FUNCTION_BLOCK SM_TableManager EXTENDS  KvalStateMachineBaseExt IMPLEMENTS I_DoorTracker
VAR_INPUT
	pStatus_bAnyTableDoorTrackTargetChanged : POINTER TO BOOL;
	cmd_bReset							: BOOL; // reset from error state
	cmd_bAbort							: BOOL; // trigger event to abort any motion.
	// Job Sync (v1.0)
    fbJobSync							: FB_JobSynchronizer;
	cmd_sJobName 						: STRING;
	cmd_sJobNameLatched					: STRING;
	// commands
	cmd_bToFenceFwd						: BOOL;
	cmd_bToFenceRev						: BOOL;
	cmd_bCrossTransferFwd				: BOOL;
	cmd_bCrossTransferRev				: BOOL;
	cmd_bInlineTransferFwd				: BOOL;
	cmd_bInlineTransferRev				: BOOL;
	cmd_bJogSlow						: BOOL;
	cmd_bManualControlEnabled			: BOOL;
	cmd_bOutputPortEnabled				: BOOL;
	cmd_bRotate							: BOOL;
	cmd_bSelfCenter						: BOOL;	
	cmd_bExternal						: BOOL;
	cmd_bInternal						: BOOL;
	
	cmd_bDoorHasNoTarget 					: BOOL;
	cmd_bInitialized 						: BOOL;
	cmd_bDoorTransferInStarted 				: BOOL;
	cmd_bDoorDataReady 						: BOOL;
	cmd_bDoorDataReadyLatched 				: BOOL;
	cmd_bNewRouteRequested 					: BOOL;	
	cmd_bReroute							: BOOL;
	cmd_bReroutePending						: BOOL;
	cmd_bNewRouteRequestedFromDoorInMachineIdle : BOOL;
	cmd_bNewRouteRequestedFromWaitForFeedout : BOOL;
	cmd_bNewRouteRequestedFromAllTargetFeedoutPortsDisabled : BOOL;
	cmd_bNewRouteRequestedFromDoorHasNoTarget : BOOL;
	cmd_bNewRouteRequestedFromWaitingForClearRoute : BOOL;
	cmd_bDoorTransferInCompleted 			: BOOL;
	cmd_bFeedinStarted 						: BOOL;
	cmd_bFeedinCompleted 					: BOOL;

	cmd_bReadyToFeedOut : BOOL;
	cmd_bDoorTransferOutStartedFromIdle 	: BOOL;
	cmd_bDoorTransferOutStarted 			: BOOL;
	cmd_bDoorTransferOutCompleted 			: BOOL;
	cmd_bFeedoutStarted 					: BOOL;
	cmd_bFeedoutCompleted 					: BOOL;
	
	cmd_iSelectedDestinationIndexLast		: UINT;
	cmd_iSelectedDestinationIndex			: UINT;
	cmd_eIncomingDoorHand					: E_DOORHAND;
	cmd_eIncomingDoorHandLast				: E_DOORHAND;
	cmd_bIncomingDoorHandValid				: BOOL;
	cmd_iSelectedDestinationIndexLatched	: UINT;
	cmd_eIncomingDoorHandLatched			: E_DOORHAND;
	
	cmd_bNewTargetFeedoutPortSelected		: BOOL;
	cmd_stNewTargetFeedoutPort				: ST_FeedoutPort;
	config_bAutoDataReady					: BOOL; // true if table is an input port and the input port is configured for 'hungry-mode' where destination index 0 is mapped to 2 or more feed-out ports. 
													// On rising edge of LH/RH input valid, 'Data Ready' input is latched automatically, instead of user needs to press the 'Data Ready' button.
													// The physical 'Data Ready' button and the 'Destination Index' switch on the control box are not needed.
													
	config_bIsInputPortEnabled				: BOOL; // true if the table's input port is enabled and can receive door data from KvalCAM's job such as destination index and doorHand.
	config_bIsConveyorTable					: BOOL; // true if it's a conveyor table (class code 235); false = auto-cross transfer table (class code 234)
	config_bCanSelfCenter					: BOOL; // true if table has the self-centering option (Option S)
	config_bCanRotate						: BOOL; // true if table has the Auto-rotate option (Option A)
	cmd_bRequestNewRoute					: BOOL;
	config_bCanFeedinFromSideA				: BOOL; // true if it's an input port and its side A is available to feed-in door.
	config_bIsBufferTable					: BOOL; // true table is a T1 option, which can only do inline-transfer and not (cross-transfer or self-center)
	
	// --- Pointers to hot connect hardware --
	config_pstHcTransferTableHardware		: POINTER TO ST_HcTable;
	config_pstHcConveyorHardware			: POINTER TO ST_HcConveyor;
	
	// each table can have either a conveyor or a cross-and-straight manager, but not both.
	smC235FeedManager						: SM_235FeedManager; // manage cross feeding of the door in and out the machine.
	smC234FeedManager						: SM_234FeedManager; // manage cross-feeding of the door in and out the machine. 
	
	smDoorDasher							: SM_DoorDasher; // a door-dasher for DTS.
	
{IF defined (noHW) OR defined (noHW_UML)}
	psmHcFeedMotor							: POINTER TO SM_KMotorVFDEtherCATi550Ext; // balvm3539 1140 RPM 1/2 HP
{ELSE}
	psmHcFeedMotor							: POINTER TO SM_KMotorVFDEtherCATi550; // balvm3539 1140 RPM 1/2 HP
{END_IF}
	
	config_tRerouteWaitTime			: TIME := T#1.0S;
	
	// feed system configs
	// these are initialized from table topology sent by KvalCAM when press Ctrl+Shift+S key combination on the Main tab:
	config_iFeedFastSpeedFPM		: UINT := 150;				// Fast Feed Speed in Feet Per Minute
	config_iFeedSlowSpeedFPM		: UINT := 50;				// Slow Feed Speed in Feet Per Minute
	config_iFeedOutSpeedFPM			: UINT := 100;				// the speed at which the system feed's out.
	config_iCrossFeedFastSpeedFPM	: UINT := 75;				// Fast CrossFeed Speed in Feet Per Minute
	config_iCrossFeedSlowSpeedFPM	: UINT := 25;				// Slow CrossFeed Speed in Feet Per Minute
	config_iTableArrayIndex					: INT;						// The array table index.
	bDoorTrackDirty							: BOOL;
END_VAR
VAR_OUTPUT
	bTableReady : BOOL; // true if the table is ready to receive door.
	bTableIsEmpty : BOOL; // true if table is empty.
	bDoorInMachine				: BOOL; // true if NOT bTableIsEmpty AND door is completely inside machine (ie, not on C234's di_C or di_D eye)
	bOkToFeedOut		: BOOL;				// depending on the direction, is it ok to feed out?
	bHasDoor			: BOOL;		// true if bDoorInMachine is true.
	
	bReadyToRotate				: BOOL;
	bOkToSelfCenter : BOOL;
	bExternal: BOOL;
	status_bMoving		: BOOL;
	
	_bAllTargetFeedoutPortsDisabled : BOOL; // true if all of the Target's feedout ports are disabled.
	bAllTargetFeedoutPortsDisabled : BOOL; // true if all of the Target's feedout ports are disabled.
	_bDoorHasNoTarget : BOOL; // true if the init seq found a door on table but no Target is assigned.
	bDoorHasNoTarget : BOOL; // true if the init seq found a door on table but no Target is assigned.
	bCurrentTargetFeedoutPortEnabled : BOOL; // true if any of the Target's feed-out port is enabled.
	bAnyCurrentTargetFeedoutPortEnabled : BOOL;
	bAllCurrentTargetFeedoutPortsEnabled : BOOL;
	bAnySourceDestinationIndexFeedoutPortEnabled : BOOL;
	
	bAnyDestinationIndexFeedoutPortEnabled : BOOL; // true if any of the feed-out port is enabled from the DestinationIndexFeedoutPortsMapping.
	bDoorInMachineIdle : BOOL;
	bDoorWaitingForFeedOut: BOOL;
	bWaitForDataReadyOrTransferredIn : BOOL;
	bDoorTransferringIn : BOOL;
	bRouteReadyWaitForFeedIn : BOOL;
	bDoorFeedingIn : BOOL;
	bDoorFeedingOut : BOOL;
	bWaitAllTablesReady : BOOL;
	bWaitingForClearRoute: BOOL;
	bRequestNewRouteComplete : BOOL;
	bFindingPath: BOOL;
END_VAR
VAR CONSTANT
END_VAR
VAR_INPUT PERSISTENT
	stDoorTrack									: ST_DoorTrack;
END_VAR
VAR PERSISTENT
	config_bManualControlEnabled				: BOOL;
END_VAR
VAR
	tonEyeBlowoffTimer							: TON;
	tofJambKickOverTimer						: TOF;
	ftrigHasDoor								: F_TRIG;
	stDoorTrackLast								: ST_DoorTrack;
	rtrigPersistentDataChanged					: R_TRIG; // triggered when any of the persistent data (feedout aligned/manual control enabled/disabled changed)	
	rtrigAutofeedOn								: R_TRIG; // rising edge of cmd_bAutofeedOn.
	ftrigAutofeedOn								: F_TRIG; // falling edge of cmd_bAutofeedOn.		
	ftrigAnyChildNotAutofeedOn					: F_TRIG; // falling edge of cmd_bAutofeedOn.
	fbVfdSetupData								: FB_VfdSetupData;
	ftrigRotateComplete							: F_TRIG; // trigger to indicate the rotate sequence is completed.
	ftrigSelfCenterComplete						: F_TRIG; // trigger to indicate the self-center sequence is completed.
	rtrigExternal								: R_TRIG;
	rtrigInternal								: R_TRIG; 
	rtrigTargetFeedoutPortsDisabled				: R_TRIG; // On rising edge, all Target table's feed-out ports were turned off by operator. 
	ftrigTargetFeedoutPortsDisabled				: F_TRIG; // On falling edge, at least 1 of the table's feed-out ports was re-enabled or operator selected a new Target feed-out port. 
	rtrigAllTargetFeedoutPortsDisabled			: R_TRIG; // Door is in-machine. On rising edge, all Target's feedout ports are disabled.
	ftrigAllTargetFeedoutPortsDisabled			: F_TRIG; // Door is in-machine. On falling edge, at least one of Target's feedout ports is enabled.
	ftrigAnyNeighboringTableBusy				: F_TRIG;
	
	rtrigDoorHasNoTarget						: R_TRIG; // On rising edge, door is detected after init but has not Target set (ie, Target = -1). Might be data persistent is corrupted.
	ftrigDoorHasNoTarget						: F_TRIG; // On falling edge, door is assigned new Target by operator.
	
	ftrigSelectedDestinationIndexChanged		: F_TRIG;
	rtrigIncomingDoorHandChanged				: R_TRIG;
	ftrigIncomingDoorHandValid					: F_TRIG;
	rtrigAutoDataReadyChanged					: R_TRIG;
	
	rtrigRequestNewRoute						: R_TRIG; // on rising edge, set cmd_bNewRouteRequested:=true to filter out stDoorTrack.Target so it does not show up in the DestinationIndex popup.
	rtrigDoorDataReady							: R_TRIG; // On rising edge while waiting for feeding out or operator selected new feed-out port, a re-route is request.
	rtrigDoorDataReadyLatched					: R_TRIG;
	ftrigDoorDataReadyLatched					: F_TRIG;
	rtrigAnyFeedoutTableEmptyAndReady			: R_TRIG;
	rtrigAnyTableWithDoorInMachineAndIdle		: R_TRIG;
	
	ftrigDoorTransferredOut						: F_TRIG;
	rtrigTableIndexNotExistInDoorTrackTargetPath		: R_TRIG;
	
	rtrigAnyTableDoorTrackTargetChanged 		: R_TRIG;
	
	rtrigAllCurrentTargetFeedoutPortsEnabled	: R_TRIG;
	ftrigAllCurrentTargetFeedoutPortsEnabled	: F_TRIG;
	
	rtrigAnyCurrentTargetFeedoutPortEnabled 	: R_TRIG;
	ftrigAnyCurrentTargetFeedoutPortEnabled 	: F_TRIG;
	
	rtrigAnyDestinationIndexFeedoutPortEnabled 	: R_TRIG;
	ftrigAnyDestinationIndexFeedoutPortEnabled 	: F_TRIG;
	rtrigDoorDasherReady 						: R_TRIG; // rising edge the door is in-machine and is ready to be transferred out. 
	rtrigRerouteAllTablesWaitingTransferredOut  : R_TRIG;
	bReadyToFeedout								: BOOL;
	rtrigReadyToFeedout							: R_TRIG; 
	ftrigReadyToFeedout							: F_TRIG;
	ftrigAnyDoorDasherBusy						: F_TRIG;
	ftrigNewRouteRequestedFromAllTargetFeedoutPortsDisabled : F_TRIG;
	ftrigNewRouteRequestedFromDoorHasNoTarget 	: F_TRIG;
	
	iFeedFastSpeedRPM		: UINT;
	iFeedSlowSpeedRPM		: UINT;
	iFeedOutSpeedRPM		: UINT;
	iCrossFeedFastSpeedRPM	: UINT;
	iCrossFeedSlowSpeedRPM	: UINT;
	bHasTrackingInfo : BOOL;
	bHasEnabledFeedoutPorts : BOOL;
	bFoundValidRoute : BOOL;
	iSourceDestinationIndexFeedoutPortsCount : UINT;
	bIsHungryModeRouting : BOOL;	
	bAnyTableBusy : BOOL;
	bAllTablesReady : BOOL;	
	bAnyNeighboringTableHasDoorAndDataReadyActive : BOOL;
	bAnyFeedoutTableEmptyAndReady: BOOL;
	bAnyNeighboringTableEmpty: BOOL;
	bAnyTableEmpty : BOOL;
	bAnyTableWithDoorHasNoTarget : BOOL;
	bSelectedDestinationIndexChanged : BOOL;
    tofSelectedDestinationIndexChangedTimer : TOF;
	bAutoDataReadyConfigChanged : BOOL;
	bAutoDataReadyConfigLast : BOOL;
	
	tonAllTablesReady	: TON;
	rtrigAllTablesReady : R_TRIG;
END_VAR

{IF defined (noHW) OR defined (noHW_UML)}
	runMachine();
{ELSE}
	readInputs();
	runMachine();
	writeOutputs();
{END_IF}

METHOD addCandidateRouteToDoorTrack
VAR_INPUT
	pstCandidateRoute : POINTER TO ST_Route;
	eTargetFeedoutSide : E_FeedoutSideType;	
END_VAR
IF pstCandidateRoute = 0 THEN
	RETURN;
END_IF

// Commented out to include duplicate table indices. This is because each duplicate table index can have up to 3 different feed-out sides, each can have
// different OutfeedDoorOrientation. 
//IF NOT isTableIndexExistInCandidateRoutes(pstCandidateRoute^.TargetTableIndex) THEN
	stDoorTrack.CandidateRoutes.CandidateRoutes[stDoorTrack.CandidateRoutes.CandidateRoutesCount] := pstCandidateRoute^;
	stDoorTrack.CandidateRoutes.CandidateRoutes[stDoorTrack.CandidateRoutes.CandidateRoutesCount].TargetFeedoutSide := eTargetFeedoutSide;
	stDoorTrack.CandidateRoutes.CandidateRoutesCount := stDoorTrack.CandidateRoutes.CandidateRoutesCount + 1;
//END_IF
END_METHOD

METHOD addSearchResultToDoorTrack
VAR_INPUT
	searchResult : ST_SearchResult;
END_VAR
stDoorTrack.SearchResults.SearchResults[stDoorTrack.SearchResults.SearchResultsCount] := searchResult;
stDoorTrack.SearchResults.SearchResultsCount := stDoorTrack.SearchResults.SearchResultsCount + 1;
END_METHOD

METHOD addToAllEnabledFeedoutPorts
VAR_INPUT
	stFeedoutPort : ST_FeedoutPort;
END_VAR
IF stDoorTrack.AllEnabledFeedoutPorts.FeedoutPortsCount >= 0 AND
	stDoorTrack.AllEnabledFeedoutPorts.FeedoutPortsCount < MAX_FEEDOUT_PORTS THEN
	stDoorTrack.AllEnabledFeedoutPorts.FeedoutPorts[stDoorTrack.AllEnabledFeedoutPorts.FeedoutPortsCount] := stFeedoutPort;
	stDoorTrack.AllEnabledFeedoutPorts.FeedoutPortsCount := stDoorTrack.AllEnabledFeedoutPorts.FeedoutPortsCount + 1;
END_IF
END_METHOD

METHOD addToRejectedFeedoutPorts
VAR_INPUT
	stFeedoutPort : ST_FeedoutPort;
END_VAR
IF stDoorTrack.RejectedFeedoutPorts.FeedoutPortsCount >= 0 AND
	stDoorTrack.RejectedFeedoutPorts.FeedoutPortsCount < MAX_FEEDOUT_PORTS THEN
	stDoorTrack.RejectedFeedoutPorts.FeedoutPorts[stDoorTrack.RejectedFeedoutPorts.FeedoutPortsCount] := stFeedoutPort;
	stDoorTrack.RejectedFeedoutPorts.FeedoutPortsCount := stDoorTrack.RejectedFeedoutPorts.FeedoutPortsCount + 1;
END_IF
END_METHOD

METHOD addToReroutableFeedoutPorts
VAR_INPUT
	stFeedoutPort : ST_FeedoutPort;
END_VAR
IF stDoorTrack.ReroutableFeedoutPorts.FeedoutPortsCount >= 0 AND
	stDoorTrack.ReroutableFeedoutPorts.FeedoutPortsCount < MAX_SEARCH_RESULTS THEN
	stDoorTrack.ReroutableFeedoutPorts.FeedoutPorts[stDoorTrack.ReroutableFeedoutPorts.FeedoutPortsCount] := stFeedoutPort;
	stDoorTrack.ReroutableFeedoutPorts.FeedoutPortsCount := stDoorTrack.ReroutableFeedoutPorts.FeedoutPortsCount + 1;
END_IF
END_METHOD

METHOD addToTargetFeedoutPorts
VAR_INPUT
	stFeedoutPort : ST_FeedoutPort;
END_VAR
IF stDoorTrack.TargetFeedoutPorts.FeedoutPortsCount >= 0 AND
	stDoorTrack.TargetFeedoutPorts.FeedoutPortsCount < MAX_FEEDOUT_PORTS THEN
	stDoorTrack.TargetFeedoutPorts.FeedoutPorts[stDoorTrack.TargetFeedoutPorts.FeedoutPortsCount] := stFeedoutPort;
	stDoorTrack.TargetFeedoutPorts.FeedoutPortsCount := stDoorTrack.TargetFeedoutPorts.FeedoutPortsCount + 1;
END_IF
END_METHOD

METHOD allChildrenAutoFeedOn : BOOL
VAR_INPUT
END_VAR
IF config_bIsConveyorTable THEN
	allChildrenAutoFeedOn := smC235FeedManager.cmd_bAutoFeedOn AND smDoorDasher.cmd_bAutofeedOn;
ELSE
	allChildrenAutoFeedOn := smC234FeedManager.cmd_bAutoFeedOn AND smDoorDasher.cmd_bAutofeedOn;
END_IF
END_METHOD

METHOD allCurrentTargetFeedoutPortsEnabled : BOOL
VAR_INPUT
END_VAR
VAR
	i : INT;
	j : INT;
	k : INT;
	stFeedoutPort : ST_FeedoutPort;
END_VAR
allCurrentTargetFeedoutPortsEnabled := TRUE; // default true to only check after Target and DestinationIndex were assigned.
IF 	stDoorTrack.DestinationIndex <> -1 
	AND stDoorTrack.TargetFeedoutPorts.FeedoutPortsCount > 0 
	THEN		
	FOR i:=0 TO stDoorTrack.TargetFeedoutPorts.FeedoutPortsCount - 1 DO
		stFeedoutPort := stDoorTrack.TargetFeedoutPorts.FeedoutPorts[i];
		IF NOT MAIN.mainStateMachine.asmTableManagers[stFeedoutPort.TableIndex].isFeedoutSideEnabled(stFeedoutPort.Side) THEN
			allCurrentTargetFeedoutPortsEnabled := FALSE;
			RETURN;
		END_IF
	END_FOR
END_IF
END_METHOD

METHOD allTablesReady : BOOL
VAR 
	i : INT;
END_VAR
allTablesReady := TRUE;

FOR i:=0 TO  MAIN.mainStateMachine.smCtrlInterface.config_stTransferTableConfig.PrimaryTable.TablesCount-1 DO
	IF NOT MAIN.mainStateMachine.smCtrlInterface.config_stTransferTableConfig.PrimaryTable.Tables[i].IsFunctionalTable THEN
		CONTINUE;
	END_IF
	
	IF  MAIN.mainStateMachine.asmTableManagers[i].bDoorFeedingIn OR
		MAIN.mainStateMachine.asmTableManagers[i].bDoorFeedingOut OR
		MAIN.mainStateMachine.asmTableManagers[i].bDoorWaitingForFeedOut OR 
		(MAIN.mainStateMachine.asmTableManagers[i].bDoorInMachineIdle AND 
		MAIN.mainStateMachine.asmTableManagers[i].stDoorTrack.Target = i) THEN
		// door is at the Target feed-out port, skip checking.
		CONTINUE;
	END_IF
	
	IF MAIN.mainStateMachine.asmTableManagers[i].status_bBusy THEN
		allTablesReady := FALSE;
		RETURN;
	END_IF
END_FOR
END_METHOD

METHOD anyChildAutofeedOn : BOOL
VAR_INPUT
END_VAR
IF config_bIsConveyorTable THEN
	anyChildAutofeedOn :=   smC235FeedManager.cmd_bAutoFeedOn OR smDoorDasher.cmd_bAutofeedOn;
ELSE
	anyChildAutofeedOn :=   smC234FeedManager.cmd_bAutoFeedOn OR smDoorDasher.cmd_bAutofeedOn;
END_IF
END_METHOD

METHOD anyChildBusy : BOOL
VAR_INPUT
END_VAR
IF config_bIsConveyorTable THEN
	anyChildBusy := smC235FeedManager.status_bBusy;
ELSE
	anyChildBusy := smC234FeedManager.status_bBusy;
END_IF
END_METHOD

METHOD anyChildExternal : BOOL
VAR_INPUT
END_VAR
IF config_bIsConveyorTable THEN
	anyChildExternal :=   smC235FeedManager.bExternal;
ELSE
	anyChildExternal :=   smC234FeedManager.bExternal;
END_IF
END_METHOD

METHOD anyCurrentTargetFeedoutPortEnabled : BOOL
VAR_INPUT
END_VAR
VAR
	i : INT;
	j : INT;
	k : INT;
	stFeedoutPort : ST_FeedoutPort;
END_VAR
anyCurrentTargetFeedoutPortEnabled := FALSE;
IF 	stDoorTrack.DestinationIndex <> -1 
	AND stDoorTrack.TargetFeedoutPorts.FeedoutPortsCount > 0 
	THEN		
	FOR i:=0 TO stDoorTrack.TargetFeedoutPorts.FeedoutPortsCount - 1 DO
		stFeedoutPort := stDoorTrack.TargetFeedoutPorts.FeedoutPorts[i];
		IF MAIN.mainStateMachine.asmTableManagers[stFeedoutPort.TableIndex].isFeedoutSideEnabled(stFeedoutPort.Side) THEN
			anyCurrentTargetFeedoutPortEnabled := TRUE;
			RETURN;
		END_IF
	END_FOR
END_IF
END_METHOD

METHOD anyDestinationIndexFeedoutPortEnabled : BOOL
VAR_INPUT
END_VAR
VAR
	i : INT;
	j : INT;
	k : INT;
	stFeedoutPort : ST_FeedoutPort;
END_VAR
anyDestinationIndexFeedoutPortEnabled := TRUE; // default true to only check after Target and DestinationIndex were assigned.
IF 	stDoorTrack.DestinationIndex <> -1 
	THEN
	// the table has a Target table, now check if any of the feed-out port is enabled from the DestinationIndexFeedoutPortsMapping.
	anyDestinationIndexFeedoutPortEnabled := FALSE;
	i := stDoorTrack.Source;
	IF MAIN.mainStateMachine.smCtrlInterface.config_stTransferTableConfig.PrimaryTable.Tables[i].DestinationsFeedoutPortsMappingConfig.DestinationsFeedoutPortsMappingsCount > 0 THEN
		FOR j:=0 TO MAIN.mainStateMachine.smCtrlInterface.config_stTransferTableConfig.PrimaryTable.Tables[i].DestinationsFeedoutPortsMappingConfig.DestinationsFeedoutPortsMappingsCount - 1 DO
			IF MAIN.mainStateMachine.smCtrlInterface.config_stTransferTableConfig.PrimaryTable.Tables[i].DestinationsFeedoutPortsMappingConfig.DestinationsFeedoutPortsMappings[j].DestinationIndex = stDoorTrack.DestinationIndex THEN
				IF MAIN.mainStateMachine.smCtrlInterface.config_stTransferTableConfig.PrimaryTable.Tables[i].DestinationsFeedoutPortsMappingConfig.DestinationsFeedoutPortsMappings[j].FeedoutPortsCount > 0 THEN
					FOR k:=0 TO MAIN.mainStateMachine.smCtrlInterface.config_stTransferTableConfig.PrimaryTable.Tables[i].DestinationsFeedoutPortsMappingConfig.DestinationsFeedoutPortsMappings[j].FeedoutPortsCount - 1 DO
						stFeedoutPort := MAIN.mainStateMachine.smCtrlInterface.config_stTransferTableConfig.PrimaryTable.Tables[i].DestinationsFeedoutPortsMappingConfig.DestinationsFeedoutPortsMappings[j].FeedoutPorts[k];
						IF MAIN.mainStateMachine.asmTableManagers[stFeedoutPort.TableIndex].isFeedoutSideEnabled(stFeedoutPort.Side) THEN
							anyDestinationIndexFeedoutPortEnabled := TRUE;
							RETURN;
						END_IF
					END_FOR
				END_IF
				EXIT;
			END_IF
		END_FOR
	END_IF
END_IF
END_METHOD

METHOD anyDoorDasherBusy : bool
VAR 
	i : INT;
END_VAR
anyDoorDasherBusy := FALSE;	
FOR i:=0 TO MAIN.mainStateMachine.smCtrlInterface.config_stTransferTableConfig.PrimaryTable.TablesCount-1 DO
	IF NOT MAIN.mainStateMachine.smCtrlInterface.config_stTransferTableConfig.PrimaryTable.Tables[i].IsFunctionalTable THEN
		CONTINUE;
	END_IF
	IF MAIN.mainStateMachine.asmTableManagers[i].smDoorDasher.status_bBusy THEN
		anyDoorDasherBusy := TRUE;
		RETURN;		
	END_IF
END_FOR
END_METHOD

METHOD anyFeedoutTableEmptyAndReady : bool
VAR 
	i : INT;
END_VAR
anyFeedoutTableEmptyAndReady := FALSE;	
FOR i:=0 TO MAIN.mainStateMachine.smCtrlInterface.config_stTransferTableConfig.PrimaryTable.TablesCount-1 DO
	IF NOT (MAIN.mainStateMachine.smCtrlInterface.config_stTransferTableConfig.PrimaryTable.Tables[i].IsFunctionalTable AND
		MAIN.mainStateMachine.smCtrlInterface.config_stTransferTableConfig.PrimaryTable.Tables[i].IsOutputPort AND 
		MAIN.mainStateMachine.smCtrlInterface.config_stTransferTableConfig.PrimaryTable.Tables[i].OutputPortEnabled) THEN
		CONTINUE;
	END_IF
	IF  //MAIN.mainStateMachine.asmTableManagers[i].bWaitForDataReadyOrTransferredIn AND
		NOT (MAIN.mainStateMachine.asmTableManagers[i].bHasDoor OR 
			MAIN.mainStateMachine.asmTableManagers[i].status_bBusy OR
			MAIN.mainStateMachine.asmTableManagers[i].cmd_bDoorDataReadyLatched) THEN
		anyFeedoutTableEmptyAndReady := TRUE;
		RETURN;		
	END_IF
END_FOR
END_METHOD

METHOD anyNeighboringTableBusy : bool
VAR 
	northNeighborIndex : INT;
	southNeighborIndex : INT;
	eastNeighborIndex : INT;
	westNeighborIndex : INT;
END_VAR
anyNeighboringTableBusy := FALSE;
northNeighborIndex := MAIN.mainStateMachine.smCtrlInterface.config_stTransferTableConfig.PrimaryTable.Tables[config_iTableArrayIndex].NeighborNorthIndex;
southNeighborIndex := MAIN.mainStateMachine.smCtrlInterface.config_stTransferTableConfig.PrimaryTable.Tables[config_iTableArrayIndex].NeighborSouthIndex;
eastNeighborIndex := MAIN.mainStateMachine.smCtrlInterface.config_stTransferTableConfig.PrimaryTable.Tables[config_iTableArrayIndex].NeighborEastIndex;
westNeighborIndex := MAIN.mainStateMachine.smCtrlInterface.config_stTransferTableConfig.PrimaryTable.Tables[config_iTableArrayIndex].NeighborWestIndex;

IF northNeighborIndex <> -1 THEN
	IF MAIN.mainStateMachine.asmTableManagers[northNeighborIndex].status_bBusy THEN
		anyNeighboringTableBusy := TRUE;
		RETURN;
	END_IF
END_IF
IF southNeighborIndex <> -1 THEN
	IF MAIN.mainStateMachine.asmTableManagers[southNeighborIndex].status_bBusy THEN
		anyNeighboringTableBusy := TRUE;
		RETURN;
	END_IF
END_IF
IF eastNeighborIndex <> -1 THEN
	IF MAIN.mainStateMachine.asmTableManagers[eastNeighborIndex].status_bBusy THEN
		anyNeighboringTableBusy := TRUE;
		RETURN;
	END_IF
END_IF
IF westNeighborIndex <> -1 THEN
	IF MAIN.mainStateMachine.asmTableManagers[westNeighborIndex].status_bBusy THEN
		anyNeighboringTableBusy := TRUE;
		RETURN;
	END_IF
END_IF
END_METHOD

METHOD anyNeighboringTableEmpty : bool
VAR 
	northNeighborIndex : INT;
	southNeighborIndex : INT;
	eastNeighborIndex : INT;
	westNeighborIndex : INT;
END_VAR
anyNeighboringTableEmpty := FALSE;
northNeighborIndex := MAIN.mainStateMachine.smCtrlInterface.config_stTransferTableConfig.PrimaryTable.Tables[config_iTableArrayIndex].NeighborNorthIndex;
southNeighborIndex := MAIN.mainStateMachine.smCtrlInterface.config_stTransferTableConfig.PrimaryTable.Tables[config_iTableArrayIndex].NeighborSouthIndex;
eastNeighborIndex := MAIN.mainStateMachine.smCtrlInterface.config_stTransferTableConfig.PrimaryTable.Tables[config_iTableArrayIndex].NeighborEastIndex;
westNeighborIndex := MAIN.mainStateMachine.smCtrlInterface.config_stTransferTableConfig.PrimaryTable.Tables[config_iTableArrayIndex].NeighborWestIndex;

IF northNeighborIndex <> -1 THEN
	IF NOT (MAIN.mainStateMachine.asmTableManagers[northNeighborIndex].bHasDoor
			) THEN
		anyNeighboringTableEmpty := TRUE;
		RETURN;
	END_IF
END_IF
IF southNeighborIndex <> -1 THEN
	IF NOT (MAIN.mainStateMachine.asmTableManagers[southNeighborIndex].bHasDoor
			) THEN
		anyNeighboringTableEmpty := TRUE;
		RETURN;
	END_IF
END_IF
IF eastNeighborIndex <> -1 THEN
	IF NOT (MAIN.mainStateMachine.asmTableManagers[eastNeighborIndex].bHasDoor
			) THEN
		anyNeighboringTableEmpty := TRUE;
		RETURN;
	END_IF
END_IF
IF westNeighborIndex <> -1 THEN
	IF NOT (MAIN.mainStateMachine.asmTableManagers[westNeighborIndex].bHasDoor
			) THEN
		anyNeighboringTableEmpty := TRUE;
		RETURN;
	END_IF
END_IF
END_METHOD

METHOD anyNeighboringTableEmptyAndNotInPath : bool
VAR 
	northNeighborIndex : INT;
	southNeighborIndex : INT;
	eastNeighborIndex : INT;
	westNeighborIndex : INT;
END_VAR
anyNeighboringTableEmptyAndNotInPath := FALSE;
northNeighborIndex := MAIN.mainStateMachine.smCtrlInterface.config_stTransferTableConfig.PrimaryTable.Tables[config_iTableArrayIndex].NeighborNorthIndex;
southNeighborIndex := MAIN.mainStateMachine.smCtrlInterface.config_stTransferTableConfig.PrimaryTable.Tables[config_iTableArrayIndex].NeighborSouthIndex;
eastNeighborIndex := MAIN.mainStateMachine.smCtrlInterface.config_stTransferTableConfig.PrimaryTable.Tables[config_iTableArrayIndex].NeighborEastIndex;
westNeighborIndex := MAIN.mainStateMachine.smCtrlInterface.config_stTransferTableConfig.PrimaryTable.Tables[config_iTableArrayIndex].NeighborWestIndex;

IF northNeighborIndex <> -1 THEN
	IF NOT (MAIN.mainStateMachine.asmTableManagers[northNeighborIndex].bHasDoor
			 OR isNeighborInTargetPath(northNeighborIndex)
			) THEN
		anyNeighboringTableEmptyAndNotInPath := TRUE;
		RETURN;
	END_IF
END_IF
IF southNeighborIndex <> -1 THEN
	IF NOT (MAIN.mainStateMachine.asmTableManagers[southNeighborIndex].bHasDoor
			 OR isNeighborInTargetPath(southNeighborIndex)
			) THEN
		anyNeighboringTableEmptyAndNotInPath := TRUE;
		RETURN;
	END_IF
END_IF
IF eastNeighborIndex <> -1 THEN
	IF NOT (MAIN.mainStateMachine.asmTableManagers[eastNeighborIndex].bHasDoor
			 OR isNeighborInTargetPath(eastNeighborIndex)
			) THEN
		anyNeighboringTableEmptyAndNotInPath := TRUE;
		RETURN;
	END_IF
END_IF
IF westNeighborIndex <> -1 THEN
	IF NOT (MAIN.mainStateMachine.asmTableManagers[westNeighborIndex].bHasDoor
			 OR isNeighborInTargetPath(westNeighborIndex)
			) THEN
		anyNeighboringTableEmptyAndNotInPath := TRUE;
		RETURN;
	END_IF
END_IF
END_METHOD

METHOD anyNeighboringTableHasDoorAndDataReadyActive : bool
VAR 
	northNeighborIndex : INT;
	southNeighborIndex : INT;
	eastNeighborIndex : INT;
	westNeighborIndex : INT;
END_VAR
anyNeighboringTableHasDoorAndDataReadyActive := FALSE;
northNeighborIndex := MAIN.mainStateMachine.smCtrlInterface.config_stTransferTableConfig.PrimaryTable.Tables[config_iTableArrayIndex].NeighborNorthIndex;
southNeighborIndex := MAIN.mainStateMachine.smCtrlInterface.config_stTransferTableConfig.PrimaryTable.Tables[config_iTableArrayIndex].NeighborSouthIndex;
eastNeighborIndex := MAIN.mainStateMachine.smCtrlInterface.config_stTransferTableConfig.PrimaryTable.Tables[config_iTableArrayIndex].NeighborEastIndex;
westNeighborIndex := MAIN.mainStateMachine.smCtrlInterface.config_stTransferTableConfig.PrimaryTable.Tables[config_iTableArrayIndex].NeighborWestIndex;

IF northNeighborIndex <> -1 THEN
	IF (MAIN.mainStateMachine.asmTableManagers[northNeighborIndex].bHasDoor AND
		MAIN.mainStateMachine.asmTableManagers[northNeighborIndex].cmd_bDoorDataReadyLatched
			) THEN
		anyNeighboringTableHasDoorAndDataReadyActive := TRUE;
		RETURN;
	END_IF
END_IF
IF southNeighborIndex <> -1 THEN
	IF (MAIN.mainStateMachine.asmTableManagers[southNeighborIndex].bHasDoor AND
		MAIN.mainStateMachine.asmTableManagers[southNeighborIndex].cmd_bDoorDataReadyLatched
			) THEN
		anyNeighboringTableHasDoorAndDataReadyActive := TRUE;
		RETURN;
	END_IF
END_IF
IF eastNeighborIndex <> -1 THEN
	IF (MAIN.mainStateMachine.asmTableManagers[eastNeighborIndex].bHasDoor AND
		MAIN.mainStateMachine.asmTableManagers[eastNeighborIndex].cmd_bDoorDataReadyLatched
			) THEN
		anyNeighboringTableHasDoorAndDataReadyActive := TRUE;
		RETURN;
	END_IF
END_IF
IF westNeighborIndex <> -1 THEN
	IF (MAIN.mainStateMachine.asmTableManagers[westNeighborIndex].bHasDoor AND
		MAIN.mainStateMachine.asmTableManagers[westNeighborIndex].cmd_bDoorDataReadyLatched
			) THEN
		anyNeighboringTableHasDoorAndDataReadyActive := TRUE;
		RETURN;
	END_IF
END_IF
END_METHOD

METHOD anySourceDestinationIndexFeedoutPortEnabled : BOOL
VAR_INPUT
	selectedDestinationIndex : INT;
END_VAR
VAR
	j : INT;
	k : INT;
	stFeedoutPort : ST_FeedoutPort;
END_VAR
anySourceDestinationIndexFeedoutPortEnabled := FALSE; 
IF MAIN.mainStateMachine.smCtrlInterface.config_stTransferTableConfig.PrimaryTable.Tables[config_iTableArrayIndex].DestinationsFeedoutPortsMappingConfig.DestinationsFeedoutPortsMappingsCount > 0 THEN
	FOR j:=0 TO MAIN.mainStateMachine.smCtrlInterface.config_stTransferTableConfig.PrimaryTable.Tables[config_iTableArrayIndex].DestinationsFeedoutPortsMappingConfig.DestinationsFeedoutPortsMappingsCount - 1 DO
		IF MAIN.mainStateMachine.smCtrlInterface.config_stTransferTableConfig.PrimaryTable.Tables[config_iTableArrayIndex].DestinationsFeedoutPortsMappingConfig.DestinationsFeedoutPortsMappings[j].FeedoutPortsCount > 0 THEN
			FOR k:=0 TO MAIN.mainStateMachine.smCtrlInterface.config_stTransferTableConfig.PrimaryTable.Tables[config_iTableArrayIndex].DestinationsFeedoutPortsMappingConfig.DestinationsFeedoutPortsMappings[j].FeedoutPortsCount - 1 DO
				IF MAIN.mainStateMachine.smCtrlInterface.config_stTransferTableConfig.PrimaryTable.Tables[config_iTableArrayIndex].DestinationsFeedoutPortsMappingConfig.DestinationsFeedoutPortsMappings[j].DestinationIndex = selectedDestinationIndex THEN
					stFeedoutPort := MAIN.mainStateMachine.smCtrlInterface.config_stTransferTableConfig.PrimaryTable.Tables[config_iTableArrayIndex].DestinationsFeedoutPortsMappingConfig.DestinationsFeedoutPortsMappings[j].FeedoutPorts[k];
					IF MAIN.mainStateMachine.asmTableManagers[stFeedoutPort.TableIndex].isFeedoutSideEnabled(stFeedoutPort.Side) THEN
						anySourceDestinationIndexFeedoutPortEnabled := TRUE;
						RETURN;
					END_IF
				END_IF
			END_FOR
		END_IF
	END_FOR
END_IF
END_METHOD

METHOD anyTableBusy : BOOL
VAR 
	i : INT;
END_VAR
anyTableBusy := FALSE;

FOR i:=0 TO  MAIN.mainStateMachine.smCtrlInterface.config_stTransferTableConfig.PrimaryTable.TablesCount-1 DO
	IF NOT MAIN.mainStateMachine.smCtrlInterface.config_stTransferTableConfig.PrimaryTable.Tables[i].IsFunctionalTable THEN
		CONTINUE;
	END_IF
	
	IF MAIN.mainStateMachine.asmTableManagers[i].status_bBusy THEN
		anyTableBusy := TRUE;
		RETURN;
	END_IF
END_FOR
END_METHOD

METHOD anyTableEmpty : BOOL
VAR 
	i : INT;
END_VAR
anyTableEmpty := FALSE;

FOR i:=0 TO  MAIN.mainStateMachine.smCtrlInterface.config_stTransferTableConfig.PrimaryTable.TablesCount-1 DO
	IF NOT MAIN.mainStateMachine.smCtrlInterface.config_stTransferTableConfig.PrimaryTable.Tables[i].IsFunctionalTable THEN
		CONTINUE;
	END_IF
	
	IF NOT MAIN.mainStateMachine.asmTableManagers[i].bHasDoor THEN
		anyTableEmpty := TRUE;
		RETURN;
	END_IF
END_FOR
END_METHOD

METHOD anyTableWithDoorHasNoTarget : BOOL
VAR 
	i : INT;
END_VAR
anyTableWithDoorHasNoTarget := FALSE;

FOR i:=0 TO MAIN.mainStateMachine.smCtrlInterface.config_stTransferTableConfig.PrimaryTable.TablesCount-1 DO
	IF NOT (MAIN.mainStateMachine.smCtrlInterface.config_stTransferTableConfig.PrimaryTable.Tables[i].IsFunctionalTable) THEN
		CONTINUE;
	END_IF
	IF MAIN.mainStateMachine.asmTableManagers[i].bDoorHasNoTarget THEN
		anyTableWithDoorHasNoTarget := TRUE;
		RETURN;
	END_IF
END_FOR
END_METHOD

METHOD autofeedOff
VAR_INPUT
END_VAR
smC234FeedManager.cmd_bAutoFeedOn := FALSE;
smC235FeedManager.cmd_bAutoFeedOn := FALSE;
smC234FeedManager.cmd_bAbort := TRUE;
smC235FeedManager.cmd_bAbort := TRUE;
smDoorDasher.cmd_bAutofeedOn := FALSE;
END_METHOD

METHOD autofeedOn
VAR_INPUT
END_VAR
smC234FeedManager.cmd_bAutoFeedOn := TRUE;
smC235FeedManager.cmd_bAutoFeedOn := TRUE;
smDoorDasher.cmd_bAutofeedOn := TRUE;
END_METHOD

METHOD blinkReadyToFeedoutSideA
VAR_INPUT
END_VAR
IF config_bIsConveyorTable THEN
	;
ELSE
	smC234FeedManager.blinkReadyToFeedoutSideA();
END_IF
END_METHOD

METHOD blinkReadyToFeedoutSideB
VAR_INPUT
END_VAR
IF config_bIsConveyorTable THEN
	;
ELSE
	smC234FeedManager.blinkReadyToFeedoutSideB();
END_IF
END_METHOD

METHOD blinkReadyToFeedoutSideC
VAR_INPUT
END_VAR
IF config_bIsConveyorTable THEN
	smC235FeedManager.blinkReadyToFeedoutSideC();
ELSE
	smC234FeedManager.blinkReadyToFeedoutSideC();
END_IF
END_METHOD

METHOD blinkReadyToFeedoutSideD
VAR_INPUT
END_VAR
IF config_bIsConveyorTable THEN
	smC235FeedManager.blinkReadyToFeedoutSideD();
ELSE
	smC234FeedManager.blinkReadyToFeedoutSideD();
END_IF
END_METHOD

METHOD blinkReadyToFeedoutSides
VAR_INPUT	
END_VAR
VAR 
	i : INT;
END_VAR
FOR i:=0 TO stDoorTrack.TargetFeedoutPorts.FeedoutPortsCount -1 DO
	IF stDoorTrack.TargetFeedoutPorts.FeedoutPorts[i].Side = E_FeedoutSideType.A THEN
		blinkReadyToFeedoutSideA();
	ELSIF stDoorTrack.TargetFeedoutPorts.FeedoutPorts[i].Side = E_FeedoutSideType.B THEN
		blinkReadyToFeedoutSideB();
	ELSIF stDoorTrack.TargetFeedoutPorts.FeedoutPorts[i].Side = E_FeedoutSideType.C THEN
		blinkReadyToFeedoutSideC();
	ELSIF stDoorTrack.TargetFeedoutPorts.FeedoutPorts[i].Side = E_FeedoutSideType.D THEN
		blinkReadyToFeedoutSideD();
	END_IF
END_FOR
END_METHOD

METHOD clearDoorTrack
VAR_INPUT
END_VAR
IF config_bNoHardwareTestMode THEN
	smC234FeedManager.di_InMachineEye := FALSE;
END_IF
stDoorTrack := stDoorTrackDefault;
stDoorTrackLast := stDoorTrackDefault;
setTableEmptyStatus(TRUE);
END_METHOD

METHOD clearDoorTrackDoorIdAndTarget
VAR_INPUT
END_VAR
stDoorTrack.DoorId := 0;
stDoorTrack.Target := -1;
stDoorTrack.TargetName := '--';
stDoorTrack.DoorRotateRequired := FALSE;
stDoorTrack.DoorWasRotated := FALSE;
stDoorTrack.DoorIsRotating := FALSE;
END_METHOD

METHOD clearLastError
VAR 
	i : INT;
END_VAR
SUPER^.clearLastError();
smC234FeedManager.clearLastError();
smC235FeedManager.clearLastError();
smDoorDasher.clearLastError();
END_METHOD

METHOD clearNextDoorId
VAR_INPUT	
END_VAR
stDoorTrack.DoorId := 0;
END_METHOD

METHOD computeDirectionalChanges : INT
VAR_INPUT
	pstPath : POINTER TO ST_PathInfo;
END_VAR
VAR
	i : INT;
	directionalChanges : INT;
	curDirection : E_Direction;
	tempDirection : E_Direction;
END_VAR
IF pstPath = 0 THEN
	computeDirectionalChanges := MAX_INT;
	RETURN;
END_IF

IF pstPath^.PathCount <= 1 THEN
	computeDirectionalChanges := 0;
	RETURN;
END_IF

curDirection := pstPath^.Path[0].Direction;

FOR i:=1 TO pstPath^.PathCount - 1 DO
	tempDirection := pstPath^.Path[i].Direction;
	IF tempDirection <> E_Direction.None AND curDirection <> tempDirection THEN
		curDirection := tempDirection;
		directionalChanges := directionalChanges + 1;
	END_IF
	
END_FOR

computeDirectionalChanges := directionalChanges;
END_METHOD

METHOD computeDoorsInPath : INT
VAR_INPUT
	pstPath : POINTER TO ST_PathInfo;
END_VAR
VAR
	i : INT;
	doorsInPath : INT;
END_VAR
IF pstPath = 0 THEN
	computeDoorsInPath := MAX_INT;
	RETURN;
END_IF

FOR i:= 0 TO pstPath^.PathCount - 1 DO
	IF MAIN.mainStateMachine.asmTableManagers[pstPath^.Path[i].TableIndex].bHasDoor THEN
		doorsInPath := doorsInPath + 1;
	END_IF
END_FOR

computeDoorsInPath := doorsInPath;
END_METHOD

// compute the score for each of the search result. The result with highest final score is selected and its target is saved in DoorTrack.Target.
METHOD computeFinalScore
VAR
	numberOfHopsWeight : LREAL;
	directionChangesWeight : LREAL;
	doorsInPathWeight : LREAL;
	numberOfHopsMin : LREAL;
	directionChangesMin : LREAL;
	doorsInPathMin : LREAL;
	hasEmptyTableInPathWeight : LREAL;
	hasIncomingDoorInPathWeight : LREAL;
	pstSearchResults : POINTER TO ST_SearchResults;
	pstSearchResult : POINTER TO ST_SearchResult;
	pstPathInfo : pointer to ST_PathInfo;
	pstSearchResultWithMaxFinalScore : POINTER TO ST_SearchResult;
	i : INT;
	target : INT;
	stRejectedFeedoutPort : ST_FeedoutPort;
	stReroutableFeedoutPort : ST_FeedoutPort;
	stTargetFeedoutPorts : ST_FeedoutPortsConfig;
	stAllEnabledFeedoutPorts : ST_FeedoutPortsConfig;
	stRejectedFeedoutPorts : ST_FeedoutPortsConfig;
	stReroutableFeedoutPorts : ST_ReroutableFeedoutPortsConfig;
	stCandidateRoutes : ST_CandidateRoutes;
	stSearchResults : ST_SearchResults;
END_VAR
pstSearchResults := ADR(stDoorTrack.SearchResults);
numberOfHopsWeight := MAIN.mainStateMachine.smCtrlInterface.config_stTransferTableConfig.PrimaryTable.PathFindingConfig.NumberHopsWeight;
directionChangesWeight := MAIN.mainStateMachine.smCtrlInterface.config_stTransferTableConfig.PrimaryTable.PathFindingConfig.DirectionalChangesWeight;
doorsInPathWeight := MAIN.mainStateMachine.smCtrlInterface.config_stTransferTableConfig.PrimaryTable.PathFindingConfig.DoorsInPathWeight;
hasEmptyTableInPathWeight := MAIN.mainStateMachine.smCtrlInterface.config_stTransferTableConfig.PrimaryTable.PathFindingConfig.HasEmptyTableInPathWeight;
hasIncomingDoorInPathWeight := MAIN.mainStateMachine.smCtrlInterface.config_stTransferTableConfig.PrimaryTable.PathFindingConfig.HasIncomingDoorInPathWeight;
stDoorTrack.RejectedFeedoutPorts.FeedoutPortsCount := 0; // Reset to 0 for counting the rejected feed-out ports for re-routing.
stDoorTrack.ReroutableFeedoutPorts.FeedoutPortsCount := 0; // Reset to 0 for counting the reroutable feed-out ports for re-routing.
bFoundValidRoute := FALSE;

FOR i := 0 TO pstSearchResults^.SearchResultsCount -1 DO
	pstSearchResult := ADR(pstSearchResults^.SearchResults[i]);
	pstPathInfo := ADR(pstSearchResult^.PathIno);
	pstSearchResult^.NumberOfHops := pstSearchResult^.PathIno.PathCount;
	pstSearchResult^.DirectionalChanges := computeDirectionalChanges(pstPathInfo);
	pstSearchResult^.DoorsInPath := computeDoorsInPath(pstPathInfo);
	pstSearchResult^.HasEmptyTableInPath := hasEmptyTableInPath(pstPathInfo);
	pstSearchResult^.HasDoorGoingOppositeDirection := hasDoorGoingOppositeDirection(pstPathInfo);
	pstSearchResult^.HasIncomingDoorInPath := hasIncomingDoorInPath(pstPathInfo);
	pstSearchResult^.HasDeadlockedDoorInPath := hasDeadlockedDoorInPath(pstPathInfo);
	pstSearchResult^.RotationRequired := doesPathRequireRotation(pstPathInfo, stDoorTrack.Source, stDoorTrack.DoorHand, pstSearchResult^.TargetFeedoutSide);
	pstSearchResult^.PathHasRotateOption := pathHasRotateOption(pstPathInfo);
END_FOR

numberOfHopsMin := minNumberOfHops(pstSearchResults);
directionChangesMin := minDirectionalChanges(pstSearchResults);
doorsInPathMin := minDoorsInPath(pstSearchResults);

FOR i := 0 TO pstSearchResults^.SearchResultsCount -1 DO
	pstSearchResult := ADR(pstSearchResults^.SearchResults[i]);
	
	pstSearchResult^.NumberOfHopsSubScore := numberOfHopsMin / pstSearchResult^.NumberOfHops * numberOfHopsWeight;
	
	IF pstSearchResult^.DirectionalChanges = 0 THEN
		pstSearchResult^.DirectionChangesSubScore := directionChangesWeight;
	ELSE
		pstSearchResult^.DirectionChangesSubScore := directionChangesMin / pstSearchResult^.DirectionalChanges * directionChangesWeight;
	END_IF
	
	IF pstSearchResult^.DoorsInPath = 0 THEN
		pstSearchResult^.DoorsInPathSubScore :=  doorsInPathWeight;
	ELSE
		pstSearchResult^.DoorsInPathSubScore :=  doorsInPathMin / pstSearchResult^.DoorsInPath * doorsInPathWeight;
	END_IF
 
	pstSearchResult^.HasEmptyTableInPathSubScore :=  BOOL_TO_INT(pstSearchResult^.HasEmptyTableInPath) * hasEmptyTableInPathWeight;
	
	pstSearchResult^.HasIncomingDoorInPathSubScore :=  BOOL_TO_INT(pstSearchResult^.HasIncomingDoorInPath) * hasIncomingDoorInPathWeight;
	
	pstSearchResult^.FinalScore := pstSearchResult^.NumberOfHopsSubScore + pstSearchResult^.DirectionChangesSubScore + pstSearchResult^.DoorsInPathSubScore + pstSearchResult^.HasEmptyTableInPathSubScore + pstSearchResult^.HasIncomingDoorInPathSubScore;
	
	IF pstSearchResult^.HasDoorGoingOppositeDirection OR
		pstSearchResult^.HasDeadlockedDoorInPath OR		
		((pstSearchResult^.RotationRequired XOR stDoorTrackLast.DoorWasRotated) AND NOT pstSearchResult^.PathHasRotateOption) 
	THEN
		IF cmd_bRequestNewRoute THEN
			stRejectedFeedoutPort.TableIndex := pstSearchResult^.PathIno.Path[pstSearchResult^.PathIno.PathCount - 1].TableIndex;
			stRejectedFeedoutPort.Side := pstSearchResult^.TargetFeedoutSide;
			addToRejectedFeedoutPorts(stRejectedFeedoutPort);
		END_IF
		CONTINUE;
	END_IF
	
	IF cmd_bRequestNewRoute THEN
		stReroutableFeedoutPort.TableIndex := pstSearchResult^.PathIno.Path[pstSearchResult^.PathIno.PathCount - 1].TableIndex;
		stReroutableFeedoutPort.Side := pstSearchResult^.TargetFeedoutSide;
		addToReroutableFeedoutPorts(stReroutableFeedoutPort);
	ELSE 	
		IF pstSearchResultWithMaxFinalScore = 0 THEN
			pstSearchResultWithMaxFinalScore := pstSearchResult;
		ELSIF pstSearchResult^.FinalScore > pstSearchResultWithMaxFinalScore^.FinalScore THEN
			pstSearchResultWithMaxFinalScore := pstSearchResult;
		END_IF
	END_IF
END_FOR

IF cmd_bRequestNewRoute THEN
	// save these before restoring to last door-track.	
	stAllEnabledFeedoutPorts := stDoorTrack.AllEnabledFeedoutPorts;
	stRejectedFeedoutPorts := stDoorTrack.RejectedFeedoutPorts;
	stReroutableFeedoutPorts := stDoorTrack.ReroutableFeedoutPorts;
	stCandidateRoutes := stDoorTrack.CandidateRoutes;
	stSearchResults := stDoorTrack.SearchResults;
	
	// restore to last door track. 
	stDoorTrack := stDoorTrackLast;
	
	// restore these for oeprator's manual rerouting.
	stDoorTrack.AllEnabledFeedoutPorts := stAllEnabledFeedoutPorts;
	stDoorTrack.RejectedFeedoutPorts := stRejectedFeedoutPorts;
	stDoorTrack.ReroutableFeedoutPorts := stReroutableFeedoutPorts;	
	stDoorTrack.CandidateRoutes := stCandidateRoutes;
	stDoorTrack.SearchResults := stSearchResults;
ELSE	
	IF pstSearchResultWithMaxFinalScore <> 0 THEN
		IF pstSearchResultWithMaxFinalScore^.PathIno.PathCount > 0 THEN
			stDoorTrack.Target := pstSearchResultWithMaxFinalScore^.PathIno.Path[pstSearchResultWithMaxFinalScore^.PathIno.PathCount - 1].TableIndex;
			stDoorTrack.TargetName := MAIN.mainStateMachine.smCtrlInterface.config_stTransferTableConfig.PrimaryTable.Tables[stDoorTrack.Target].Name;
			stDoorTrack.TargetPath := pstSearchResultWithMaxFinalScore^.PathIno;
			stDoorTrack.TargetFeedoutSide := pstSearchResultWithMaxFinalScore^.TargetFeedoutSide;
			stDoorTrack.DoorRotateRequired := pstSearchResultWithMaxFinalScore^.RotationRequired;
			stDoorTrack.DoorWasRotated := stDoorTrackLast.DoorWasRotated;
			stDoorTrack.HasEmptyTableInPath := pstSearchResultWithMaxFinalScore^.HasEmptyTableInPath;
			stDoorTrack.HasDoorGoingOppositeDirection := pstSearchResultWithMaxFinalScore^.HasDoorGoingOppositeDirection;
			stDoorTrack.HasIncomingDoorInPath := pstSearchResultWithMaxFinalScore^.HasIncomingDoorInPath;
			stDoorTrack.HasDeadlockedDoorInPath := pstSearchResultWithMaxFinalScore^.HasDeadlockedDoorInPath;
		END_IF
	ELSE
		// Failed to find new route. Set to default to clear TargetDoorTrackInfo on HMI.
		stDoorTrack := stDoorTrackDefault;
	END_IF
END_IF

IF cmd_bNewRouteRequestedFromDoorHasNoTarget AND stDoorTrack.Target = -1 THEN
	stDoorTrack.TargetFeedoutPorts := stAllEnabledFeedoutPorts;
ELSE
	bFoundValidRoute := stDoorTrack.Target <> -1 AND stDoorTrack.TargetPath.PathCount > 0;
	IF NOT bFoundValidRoute THEN
		stTargetFeedoutPorts := stDoorTrack.TargetFeedoutPorts;
		// restore to last door track. 
		stDoorTrack := stDoorTrackLast;		
		stDoorTrack.TargetFeedoutPorts := stTargetFeedoutPorts;
	END_IF
END_IF
END_METHOD

METHOD currentTargetFeedoutPortEnabled : BOOL
VAR_INPUT
END_VAR
VAR
	i : INT;
	j : INT;
	k : INT;
	stFeedoutPort : ST_FeedoutPort;
END_VAR
currentTargetFeedoutPortEnabled := TRUE; // default true to only check after Target and DestinationIndex were assigned.
IF 	stDoorTrack.DestinationIndex <> -1 THEN
	// the table has a Target table, now check if any of the feed-out port is enabled.
	currentTargetFeedoutPortEnabled := FALSE;
	i := stDoorTrack.Source;
	IF MAIN.mainStateMachine.smCtrlInterface.config_stTransferTableConfig.PrimaryTable.Tables[i].DestinationsFeedoutPortsMappingConfig.DestinationsFeedoutPortsMappingsCount > 0 THEN
		FOR j:=0 TO MAIN.mainStateMachine.smCtrlInterface.config_stTransferTableConfig.PrimaryTable.Tables[i].DestinationsFeedoutPortsMappingConfig.DestinationsFeedoutPortsMappingsCount - 1 DO
			IF MAIN.mainStateMachine.smCtrlInterface.config_stTransferTableConfig.PrimaryTable.Tables[i].DestinationsFeedoutPortsMappingConfig.DestinationsFeedoutPortsMappings[j].DestinationIndex = stDoorTrack.DestinationIndex THEN
				IF MAIN.mainStateMachine.smCtrlInterface.config_stTransferTableConfig.PrimaryTable.Tables[i].DestinationsFeedoutPortsMappingConfig.DestinationsFeedoutPortsMappings[j].FeedoutPortsCount > 0 THEN
					FOR k:=0 TO MAIN.mainStateMachine.smCtrlInterface.config_stTransferTableConfig.PrimaryTable.Tables[i].DestinationsFeedoutPortsMappingConfig.DestinationsFeedoutPortsMappings[j].FeedoutPortsCount - 1 DO
						stFeedoutPort := MAIN.mainStateMachine.smCtrlInterface.config_stTransferTableConfig.PrimaryTable.Tables[i].DestinationsFeedoutPortsMappingConfig.DestinationsFeedoutPortsMappings[j].FeedoutPorts[k];
						IF stDoorTrack.Target = stFeedoutPort.TableIndex AND 
							stDoorTrack.TargetFeedoutSide = stFeedoutPort.Side AND 
							MAIN.mainStateMachine.asmTableManagers[stFeedoutPort.TableIndex].isFeedoutSideEnabled(stFeedoutPort.Side) THEN
							currentTargetFeedoutPortEnabled := TRUE;
							RETURN;
						END_IF
					END_FOR
				END_IF
				EXIT;
			END_IF
		END_FOR
	END_IF
END_IF
END_METHOD

METHOD doesPathRequireRotation : BOOL
VAR_INPUT
	pstPath : POINTER TO ST_PathInfo;
	iOriginalSource : INT; // the original table index where the door first fed in.
	eDoorHand : E_DOORHAND;
	eTargetFeedoutSide : E_FeedoutSideType;
END_VAR
VAR
	targetTableIndex : INT;
	sourceBypassInfeedSideA_IsLockEdgeRightOfAB : BOOL;
	sourceDoorOrientationConfig : ST_DoorOrientationConfig;
	targetDoorOrientationConfig : ST_DoorOrientationConfig;
	sourceDoorMachineOrientation : ST_DoorMachineOrientation;
	targetDoorMachineOrientation : ST_DoorMachineOrientation;
	isSourceAndTargetDoorMachineOrientationMatched : BOOL;
END_VAR
doesPathRequireRotation := FALSE;
IF pstPath = 0 THEN	
	RETURN;
END_IF

targetTableIndex := pstPath^.Path[pstPath^.PathCount - 1].TableIndex;
sourceDoorOrientationConfig := MAIN.mainStateMachine.smCtrlInterface.config_stTransferTableConfig.PrimaryTable.Tables[iOriginalSource].InOutfeedDoorOrientationConfig.InfeedSideA;
sourceBypassInfeedSideA_IsLockEdgeRightOfAB := MAIN.mainStateMachine.smCtrlInterface.config_stTransferTableConfig.PrimaryTable.Tables[iOriginalSource].InOutfeedDoorOrientationConfig.BypassInfeedSideA_IsLockEdgeRightOfAB;

IF eTargetFeedoutSide = E_FeedoutSideType.A THEN
	targetDoorOrientationConfig := MAIN.mainStateMachine.smCtrlInterface.config_stTransferTableConfig.PrimaryTable.Tables[targetTableIndex].InOutfeedDoorOrientationConfig.OutfeedSideA;
ELSIF eTargetFeedoutSide = E_FeedoutSideType.B THEN
	targetDoorOrientationConfig := MAIN.mainStateMachine.smCtrlInterface.config_stTransferTableConfig.PrimaryTable.Tables[targetTableIndex].InOutfeedDoorOrientationConfig.OutfeedSideB;
ELSIF eTargetFeedoutSide = E_FeedoutSideType.C THEN
	targetDoorOrientationConfig := MAIN.mainStateMachine.smCtrlInterface.config_stTransferTableConfig.PrimaryTable.Tables[targetTableIndex].InOutfeedDoorOrientationConfig.OutfeedSideC;
ELSIF eTargetFeedoutSide = E_FeedoutSideType.D THEN
	targetDoorOrientationConfig := MAIN.mainStateMachine.smCtrlInterface.config_stTransferTableConfig.PrimaryTable.Tables[targetTableIndex].InOutfeedDoorOrientationConfig.OutfeedSideD;
END_IF

IF eDoorHand = E_DOORHAND.DOORHAND_LEFT THEN
	sourceDoorMachineOrientation := sourceDoorOrientationConfig.LeftHand;
	targetDoorMachineOrientation := targetDoorOrientationConfig.LeftHand;
ELSIF eDoorHand = E_DOORHAND.DOORHAND_RIGHT THEN
	sourceDoorMachineOrientation := sourceDoorOrientationConfig.RightHand;
	targetDoorMachineOrientation := targetDoorOrientationConfig.RightHand;
ELSIF eDoorHand = E_DOORHAND.DOORHAND_LEFT_REVERSE THEN
	sourceDoorMachineOrientation := sourceDoorOrientationConfig.LeftHandReverse;
	targetDoorMachineOrientation := targetDoorOrientationConfig.LeftHandReverse;
ELSIF eDoorHand = E_DOORHAND.DOORHAND_RIGHT_REVERSE THEN
	sourceDoorMachineOrientation := sourceDoorOrientationConfig.RightHandReverse;
	targetDoorMachineOrientation := targetDoorOrientationConfig.RightHandReverse;
END_IF
isSourceAndTargetDoorMachineOrientationMatched := 
	(sourceBypassInfeedSideA_IsLockEdgeRightOfAB OR 
	(sourceDoorMachineOrientation.IsLockEdgeRightOfAB = targetDoorMachineOrientation.IsLockEdgeRightOfAB)) AND
	sourceDoorMachineOrientation.IsTopEdgeOnASide = targetDoorMachineOrientation.IsTopEdgeOnASide;
doesPathRequireRotation := NOT isSourceAndTargetDoorMachineOrientationMatched;
END_METHOD

METHOD doState
CASE (machineState) OF	
	TABLEMANAGER_DISABLED:
		IF bFirstPass THEN
			downstream.setAllDownstreamDisabled();
			status_bBusy := FALSE;
			bError := FALSE;
			status_bReady := FALSE;
			cmd_bAutoFeedOn := FALSE;
			bExternal := FALSE;
			setJobProcessingPhase(E_JobProcessingPhases.JOB_PHASE_NOT_ACCEPTING);
		END_IF
                
	TABLEMANAGER_ENABLING:
		downstream.setAllDownstreamEnabled();
		IF downstream.status_bDownstreamAllReady THEN
			machineState := TABLEMANAGER_AUTOFEED_OFF;
		END_IF

	TABLEMANAGER_INLINE_JOGGING:
		status_bBusy := TRUE;
		smC234FeedManager.cmd_bInlineTransferFwd := cmd_bInlineTransferFwd;
		smC234FeedManager.cmd_bInlineTransferRev := cmd_bInlineTransferRev;
		smC234FeedManager.cmd_bJogSlow := cmd_bJogSlow;
		IF NOT (cmd_bInlineTransferFwd OR cmd_bInlineTransferRev) THEN
			machineState := TABLEMANAGER_AUTOFEED_OFF;
		END_IF
		
	TABLEMANAGER_CROSS_JOGGING:
		status_bBusy := TRUE;
		IF config_bIsConveyorTable THEN
			smC235FeedManager.cmd_bCrossTransferFwd := cmd_bCrossTransferFwd;
			smC235FeedManager.cmd_bCrossTransferRev := cmd_bCrossTransferRev;
			smC235FeedManager.cmd_bJogSlow := cmd_bJogSlow;
		ELSE
			smC234FeedManager.cmd_bCrossTransferFwd := cmd_bCrossTransferRev;
			smC234FeedManager.cmd_bCrossTransferRev := cmd_bCrossTransferFwd;
			smC234FeedManager.cmd_bJogSlow := cmd_bJogSlow;
		END_IF
		IF NOT (cmd_bCrossTransferFwd OR cmd_bCrossTransferRev) THEN
			machineState := TABLEMANAGER_AUTOFEED_OFF;
		END_IF
		
	TABLEMANAGER_TO_FENCE_JOGGING:
		status_bBusy := TRUE;
		smC234FeedManager.cmd_bToFenceFwd := cmd_bToFenceRev;
		smC234FeedManager.cmd_bToFenceRev := cmd_bToFenceFwd;
		smC234FeedManager.cmd_bJogSlow := cmd_bJogSlow;
		
		IF NOT (cmd_bToFenceFwd OR cmd_bToFenceRev) THEN
			machineState := TABLEMANAGER_AUTOFEED_OFF;
		END_IF
	
	TABLEMANAGER_ROTATE:
		IF bFirstPass THEN
			status_bBusy := TRUE;
			smC234FeedManager.cmd_bRotate := TRUE;
		END_IF
		ftrigRotateComplete(CLK:=smC234FeedManager.status_bBusy);
		IF ftrigRotateComplete.Q THEN
			machineState := TABLEMANAGER_AUTOFEED_OFF;
		END_IF
		
	TABLEMANAGER_SELF_CENTER:
		IF bFirstPass THEN
			status_bBusy := TRUE;
			smC234FeedManager.cmd_bSelfCenter := TRUE;
		END_IF
		ftrigSelfCenterComplete(CLK:=smC234FeedManager.status_bBusy);
		IF ftrigSelfCenterComplete.Q THEN
			machineState := TABLEMANAGER_AUTOFEED_OFF;
		END_IF
		
	TABLEMANAGER_AUTOFEED_OFF:
		IF bFirstPass THEN
			status_bBusy := FALSE;
			status_bReady := TRUE;
			bExternal := FALSE;
			cmd_bInitialized := FALSE;
			bFindingPath := FALSE;
			cmd_bRequestNewRoute := FALSE;
			setReadyToFeedoutSides(FALSE);
			setJobProcessingPhase(E_JobProcessingPhases.JOB_PHASE_NOT_ACCEPTING);
		END_IF

		IF cmd_bSelfCenter AND
			bOkToSelfCenter AND
			config_bCanSelfCenter AND
			cmd_bManualControlEnabled THEN
			machineState := TABLEMANAGER_SELF_CENTER;
		ELSIF cmd_bRotate AND
			bReadyToRotate AND
			config_bCanRotate AND
			cmd_bManualControlEnabled THEN
			machineState := TABLEMANAGER_ROTATE;
		ELSIF (cmd_bInlineTransferFwd OR cmd_bInlineTransferRev) AND cmd_bManualControlEnabled THEN
			machineState := TABLEMANAGER_INLINE_JOGGING;
		ELSIF (cmd_bCrossTransferFwd OR cmd_bCrossTransferRev) AND 
				(config_bIsConveyorTable OR NOT config_bIsBufferTable) AND 
				cmd_bManualControlEnabled THEN
			machineState := TABLEMANAGER_CROSS_JOGGING;	
		ELSIF (cmd_bToFenceFwd OR cmd_bToFenceRev) AND
				NOT (config_bIsBufferTable OR config_bIsConveyorTable) AND
				cmd_bManualControlEnabled THEN
			machineState := TABLEMANAGER_TO_FENCE_JOGGING;
		ELSIF cmd_bAutoFeedOn THEN
			machineState := TABLEMANAGER_AUTOFEED_ON;		
		END_IF
		
	TABLEMANAGER_AUTOFEED_ON:
		IF bFirstPass THEN			
			status_bBusy := FALSE;
			bExternal := FALSE;
			cmd_bRequestNewRoute := FALSE;
			cmd_bDoorHasNoTarget := FALSE;
			setJobProcessingPhase(E_JobProcessingPhases.JOB_PHASE_NOT_ACCEPTING);
		ELSE
			IF cmd_bInitialized THEN
				machineState := TABLEMANAGER_DOOR_TRACKER_START;
			ELSIF NOT cmd_bAutoFeedOn THEN
				machineState := TABLEMANAGER_AUTOFEED_OFF;
			END_IF
		END_IF
		
	TABLEMANAGER_DOOR_TRACKER_START:
		IF bFirstPass THEN			
			setReadyToFeedoutSides(FALSE);	
			setJobProcessingPhase(E_JobProcessingPhases.JOB_PHASE_NOT_ACCEPTING);
		END_IF
		
		IF cmd_bRequestNewRoute THEN
			machineState := TABLEMANAGER_DOOR_TRACKER_FINDPATH_INIT;
		ELSIF cmd_bNewTargetFeedoutPortSelected THEN
			machineState := TABLEMANAGER_DOOR_TRACKER_FINDPATH_INIT;
		ELSIF bHasDoor AND NOT bAnyCurrentTargetFeedoutPortEnabled THEN
			machineState := TABLEMANAGER_DOOR_TRACKER_FINDPATH_INIT;
		ELSIF bHasDoor THEN
			machineState := TABLEMANAGER_DOOR_TRACKER_DOOR_IN_MACHINE_IDLE;
		ELSIF cmd_bNext THEN
			machineState := TABLEMANAGER_DOOR_TRACKER_WAIT_FOR_DATA_READY_OR_TRANSFERRED_IN;
		END_IF

	TABLEMANAGER_DOOR_TRACKER_WAIT_FOR_DATA_READY_OR_TRANSFERRED_IN:
		IF bFirstPass THEN
			cmd_bRequestNewRoute := FALSE;
			cmd_bNewTargetFeedoutPortSelected := FALSE;
			cmd_bNewRouteRequested := FALSE;
			initDoorTrack();
			resetDoorTrack();
			clearDoorTrackDoorIdAndTarget();
			setJobProcessingPhase(E_JobProcessingPhases.JOB_PHASE_NONE_PENDING);	
		END_IF
		IF cmd_bDoorDataReadyLatched THEN
			machineState := TABLEMANAGER_DOOR_TRACKER_FINDPATH_INIT;
		ELSIF cmd_bDoorTransferInStarted THEN
			machineState := TABLEMANAGER_DOOR_TRACKER_TRANSFERRING_IN;
		END_IF

	TABLEMANAGER_DOOR_TRACKER_TRANSFERRING_IN:
		IF bFirstPass THEN
			;
		END_IF
		IF cmd_bDoorTransferInCompleted THEN
			machineState := TABLEMANAGER_DOOR_TRACKER_DOOR_IN_MACHINE_IDLE;
		END_IF
	
	TABLEMANAGER_DOOR_TRACKER_ROUTE_READY_WAIT_FOR_FEED_IN:
		IF bFirstPass THEN
			clearNextDoorId();
			setJobProcessingPhase(E_JobProcessingPhases.JOB_PHASE_PENDING);
		ELSE
			cmd_bReroute := rtrigIncomingDoorHandChanged.Q;
			IF cmd_bReroute THEN
				cmd_bReroute := FALSE;
				machineState := TABLEMANAGER_DOOR_TRACKER_FINDPATH_INIT;
			ELSIF rtrigTargetFeedoutPortsDisabled.Q THEN
				machineState := TABLEMANAGER_DOOR_TRACKER_FINDPATH_INIT;
			ELSIF NOT cmd_bDoorDataReadyLatched THEN
				machineState := TABLEMANAGER_DOOR_TRACKER_WAIT_FOR_DATA_READY_OR_TRANSFERRED_IN;			
			ELSIF cmd_bFeedinStarted THEN
				machineState := TABLEMANAGER_DOOR_TRACKER_DOOR_FEEDING_IN;
			END_IF
		END_IF
		
	TABLEMANAGER_DOOR_TRACKER_DOOR_FEEDING_IN:
		IF bFirstPass THEN
			setNextDoorId();
			iSourceDestinationIndexFeedoutPortsCount := getSourceAndDestinationIndexFeedoutPortsCount();
			bIsHungryModeRouting := iSourceDestinationIndexFeedoutPortsCount > 1;
			setJobProcessingPhase(E_JobProcessingPhases.JOB_PHASE_PRE_PROCESSING);
		ELSE
			IF cmd_bFeedinCompleted THEN
				bAnyFeedoutTableEmptyAndReady := anyFeedoutTableEmptyAndReady();
				IF bIsHungryModeRouting AND (cmd_bDoorDataReadyLatched OR bAnyFeedoutTableEmptyAndReady) 
				THEN
					machineState := TABLEMANAGER_DOOR_TRACKER_FINDPATH_INIT;
				ELSE
					machineState := TABLEMANAGER_DOOR_TRACKER_DOOR_IN_MACHINE_IDLE;
				END_IF
			END_IF
		END_IF
		
	TABLEMANAGER_DOOR_TRACKER_DOOR_IN_MACHINE_IDLE:
		IF bFirstPass THEN
			cmd_bRequestNewRoute := FALSE;
			cmd_bNewTargetFeedoutPortSelected := FALSE;
			cmd_bDoorTransferOutStarted := FALSE;
			cmd_bDoorTransferOutStartedFromIdle := FALSE;
			iSourceDestinationIndexFeedoutPortsCount := getSourceAndDestinationIndexFeedoutPortsCount();
			bIsHungryModeRouting := iSourceDestinationIndexFeedoutPortsCount > 1;
			setReadyToFeedoutSides(FALSE);
			rtrigDoorDasherReady(CLK:=FALSE);
			rtrigAnyFeedoutTableEmptyAndReady(CLK:=FALSE);
			setJobProcessingPhase(E_JobProcessingPhases.JOB_PHASE_PROCESSING);
		ELSE
			IF rtrigDoorDataReadyLatched.Q AND bIsHungryModeRouting THEN
				rerouteAllTablesWaitingTransferredOut();
			END_IF 		
			

			bAnyNeighboringTableEmpty := anyNeighboringTableEmpty();
			bAnyFeedoutTableEmptyAndReady := anyFeedoutTableEmptyAndReady();
			bAnyNeighboringTableHasDoorAndDataReadyActive := anyNeighboringTableHasDoorAndDataReadyActive();
			
			rtrigAnyFeedoutTableEmptyAndReady(CLK:=	bIsHungryModeRouting AND
													( 
													// Do not handle this case. For SN6, this causes door to move around T2 and T3 if T1's Data Ready Latch is active.
													// T5 just fed out door, T4 has door.
													//(bAnyFeedoutTableEmptyAndReady AND NOT stDoorTrack.HasIncomingDoorInPath) OR 
				
													(bAnyNeighboringTableEmpty AND bAnyNeighboringTableHasDoorAndDataReadyActive) OR
													
													// Only apply to input table.  If the Data Ready Latch is on while the the neighboring table's DoorDasher seq
													// is running, the door dasher seq of this current table might not allow to run. So this
													// check will look for an empty neighboring table periodically to move door out and clear for new incoming door. 
													(cmd_bDoorDataReadyLatched AND bAnyNeighboringTableEmpty))
													
													AND
    
													NOT status_bBusy AND
													
													// Prevent rapidly triggering reroute by waiting 1 sec before looking for an empty feed-out table to route the door to.
													tTimeInState>T#1.0S
												);
			IF rtrigAnyFeedoutTableEmptyAndReady.Q THEN
				cmd_bReroute := TRUE;
			END_IF	
				

						
			rtrigDoorDasherReady(CLK:= 
				NOT bReadyToFeedout AND
				(rtrigAnyTableDoorTrackTargetChanged.Q OR		
				NOT status_bBusy)
				);

			IF rtrigReadyToFeedout.CLK THEN
				machineState := TABLEMANAGER_DOOR_TRACKER_WAIT_FOR_FEED_OUT;			
			ELSIF rtrigTableIndexNotExistInDoorTrackTargetPath.CLK THEN
				machineState := TABLEMANAGER_DOOR_TRACKER_FINDPATH_INIT;
			ELSIF ftrigAllCurrentTargetFeedoutPortsEnabled.Q THEN
				machineState := TABLEMANAGER_DOOR_TRACKER_FINDPATH_INIT;
			ELSIF cmd_bRequestNewRoute THEN
				cmd_bNewRouteRequestedFromDoorInMachineIdle := TRUE;
				machineState := TABLEMANAGER_DOOR_TRACKER_FINDPATH_INIT;
			ELSIF cmd_bNewTargetFeedoutPortSelected THEN
				machineState := TABLEMANAGER_DOOR_TRACKER_FINDPATH_INIT;
			ELSIF cmd_bDoorTransferOutStartedFromIdle THEN
				machineState := TABLEMANAGER_DOOR_TRACKER_TRANSFERRING_OUT;			
			ELSIF cmd_bReroute AND bIsHungryModeRouting THEN
				cmd_bReroute := FALSE;				
				machineState := TABLEMANAGER_DOOR_TRACKER_FINDPATH_INIT;
			ELSIF rtrigDoorDasherReady.Q OR (NOT bIsHungryModeRouting AND rtrigDoorDasherReady.CLK) THEN
				smDoorDasher.doorDash();
			END_IF			
		END_IF
		
	TABLEMANAGER_DOOR_TRACKER_WAIT_FOR_FEED_OUT:
		IF bFirstPass THEN
			cmd_bRequestNewRoute := FALSE;
			cmd_bNewTargetFeedoutPortSelected := FALSE;
			cmd_bDoorTransferOutStarted := FALSE;
			cmd_bDoorTransferOutStartedFromIdle := FALSE;
			iSourceDestinationIndexFeedoutPortsCount := getSourceAndDestinationIndexFeedoutPortsCount();
			bIsHungryModeRouting := iSourceDestinationIndexFeedoutPortsCount > 1;
			setReadyToFeedoutSides(FALSE);
			rtrigAnyFeedoutTableEmptyAndReady(CLK:=FALSE);
		END_IF
		
		blinkReadyToFeedoutSides();
		bAnyTableEmpty := anyTableEmpty();
		bAnyNeighboringTableEmpty := anyNeighboringTableEmpty();
		bAnyFeedoutTableEmptyAndReady := anyFeedoutTableEmptyAndReady();
		bAnyTableWithDoorHasNoTarget := anyTableWithDoorHasNoTarget();
		rtrigAnyFeedoutTableEmptyAndReady(CLK:=
			(bAnyNeighboringTableEmpty OR bAnyFeedoutTableEmptyAndReady) AND
				cmd_bDoorDataReadyLatched AND
				NOT bAnyTableWithDoorHasNoTarget
			);
				
		IF 
			bIsHungryModeRouting AND // true if source+destination index feedout ports count > 1			
			(rtrigDoorDataReadyLatched.Q OR 
			rtrigAnyFeedoutTableEmptyAndReady.Q OR 
			
			// Data-ready latch is active. 
			// Periodically send out reroute request to all tables with doors. 
			(cmd_bDoorDataReadyLatched AND 
			tTimeInState>T#1.0S AND 
			(bAnyTableEmpty
			))) 
			THEN
			rerouteAllTablesWaitingTransferredOut();
			cmd_bReroute := TRUE;
		END_IF 
		
		IF ftrigReadyToFeedout.Q THEN
			machineState := TABLEMANAGER_DOOR_TRACKER_DOOR_IN_MACHINE_IDLE;
		ELSIF cmd_bReroute AND bIsHungryModeRouting THEN
			cmd_bReroute := FALSE;
			machineState := TABLEMANAGER_DOOR_TRACKER_FINDPATH_INIT;
		ELSIF ftrigAllCurrentTargetFeedoutPortsEnabled.Q THEN
			machineState := TABLEMANAGER_DOOR_TRACKER_FINDPATH_INIT;
		ELSIF cmd_bRequestNewRoute THEN
			cmd_bNewRouteRequestedFromWaitForFeedout := TRUE;
			machineState := TABLEMANAGER_DOOR_TRACKER_FINDPATH_INIT;
		ELSIF cmd_bNewTargetFeedoutPortSelected THEN
			machineState := TABLEMANAGER_DOOR_TRACKER_FINDPATH_INIT;
		ELSIF cmd_bFeedoutStarted THEN
			machineState := TABLEMANAGER_DOOR_TRACKER_DOOR_FEEDING_OUT;
		ELSIF cmd_bDoorTransferOutStarted THEN
			machineState := TABLEMANAGER_DOOR_TRACKER_TRANSFERRING_OUT;
		END_IF
	
	TABLEMANAGER_DOOR_TRACKER_DOOR_FEEDING_OUT:
		IF bFirstPass THEN
			setReadyToFeedoutSides(FALSE);
			setReadyToFeedoutSide(TRUE);
			setJobProcessingPhase(E_JobProcessingPhases.JOB_PHASE_POST_PROCESSING);
		END_IF
		IF cmd_bFeedoutCompleted THEN
			machineState := TABLEMANAGER_DOOR_TRACKER_WAIT_ALL_TABLES_READY;
		END_IF
		
	TABLEMANAGER_DOOR_TRACKER_WAIT_ALL_TABLES_READY:
		IF bFirstPass THEN
			tonAllTablesReady(IN:=FALSE, PT:=config_tRerouteWaitTime);
			rtrigAllTablesReady(CLK:=FALSE);
		END_IF
		bAllTablesReady := allTablesReady();
		tonAllTablesReady(IN:=bAllTablesReady);
		rtrigAllTablesReady(CLK:=tonAllTablesReady.Q);
		IF rtrigAllTablesReady.Q THEN
			IF NOT bHasDoor THEN
				// while waiting for all tables to be ready, a new door might be transferred in from the feed-in port (ie, SN6, T1->T5).
				// So only send reroute request to all tables with 'Door-In-Machine' state if this table has no door.
				rerouteAllTablesWaitingTransferredOut();
			END_IF
			machineState := TABLEMANAGER_DOOR_TRACKER_COMPLETE;
		END_IF
		
	TABLEMANAGER_DOOR_TRACKER_TRANSFERRING_OUT:        
		IF bFirstPass THEN
			setReadyToFeedoutSides(FALSE);
			ftrigDoorTransferredOut(CLK:=FALSE);
			setJobProcessingPhase(E_JobProcessingPhases.JOB_PHASE_POST_PROCESSING);
		ELSE
			ftrigDoorTransferredOut(CLK:=smDoorDasher.status_bBusy);
			IF ftrigDoorTransferredOut.Q THEN
				machineState := TABLEMANAGER_DOOR_TRACKER_COMPLETE;
			END_IF
		END_IF

	TABLEMANAGER_DOOR_TRACKER_COMPLETE:        
		IF bFirstPass THEN			
			setJobProcessingPhase(E_JobProcessingPhases.JOB_PHASE_FINISHED);
			IF config_bNoHardwareTestMode THEN
			   smC234FeedManager.di_InMachineEye := FALSE;
			END_IF			
		END_IF
		IF cmd_bNext THEN
			machineState := TABLEMANAGER_DOOR_TRACKER_START;		
		END_IF
		
	TABLEMANAGER_DOOR_TRACKER_FINDPATH_INIT:
		IF bFirstPass THEN			
			bFindingPath := TRUE;
			initDoorTrack();
			setReadyToFeedoutSides(FALSE);
		ELSIF cmd_bNext THEN
			IF bHasDoor AND stDoorTrack.Source <> -1 THEN
				machineState := TABLEMANAGER_DOOR_TRACKER_FINDPATH_FIND_ENABLED_FEEDOUT_PORTS;
			ELSE
				machineState := TABLEMANAGER_DOOR_TRACKER_FINDPATH_RESET;
			END_IF
		END_IF
		
	TABLEMANAGER_DOOR_TRACKER_FINDPATH_RESET:
		IF bFirstPass THEN
			resetDoorTrack();
		ELSIF cmd_bNext THEN
			machineState := TABLEMANAGER_DOOR_TRACKER_FINDPATH_FIND_ENABLED_FEEDOUT_PORTS;
		END_IF
		
	TABLEMANAGER_DOOR_TRACKER_FINDPATH_FIND_ENABLED_FEEDOUT_PORTS:
		IF bFirstPass THEN
			bHasEnabledFeedoutPorts := findAllEnabledFeedoutPorts();
		ELSIF cmd_bNext THEN
			IF bHasEnabledFeedoutPorts THEN
				machineState := TABLEMANAGER_DOOR_TRACKER_FINDPATH_FIND_CANDIDATE_ROUTES;
			ELSIF cmd_bNewRouteRequested THEN
				// restore to last door track. 
				stDoorTrack := stDoorTrackLast;
				machineState := TABLEMANAGER_DOOR_TRACKER_FINDPATH_COMPLETE;
			ELSE
				machineState := TABLEMANAGER_DOOR_TRACKER_FINDPATH_WAITING_FOR_CLEAR_ROUTE;
			END_IF
		END_IF
		
	TABLEMANAGER_DOOR_TRACKER_FINDPATH_WAITING_FOR_CLEAR_ROUTE:
		IF bFirstPass THEN
			bFindingPath := FALSE;
			cmd_bRequestNewRoute := FALSE;	
			cmd_bNewTargetFeedoutPortSelected := FALSE;
			// restore to last door track. 
			stDoorTrack := stDoorTrackLast;
			stDoorTrack.Target := -1;
			stDoorTrack.TargetName := '--';
		ELSE
			IF NOT cmd_bDoorDataReadyLatched THEN
				machineState := TABLEMANAGER_DOOR_TRACKER_FINDPATH_COMPLETE;
			ELSIF cmd_bRequestNewRoute THEN
				machineState := TABLEMANAGER_DOOR_TRACKER_FINDPATH_INIT;
				cmd_bNewRouteRequestedFromWaitingForClearRoute:=TRUE;
			ELSIF cmd_bNewTargetFeedoutPortSelected THEN
				machineState := TABLEMANAGER_DOOR_TRACKER_FINDPATH_INIT;
			ELSIF cmd_bRetry THEN
				machineState := TABLEMANAGER_DOOR_TRACKER_FINDPATH_INIT;
			END_IF
		END_IF
		
	TABLEMANAGER_DOOR_TRACKER_FINDPATH_FIND_CANDIDATE_ROUTES:
		IF bFirstPass THEN
			findAllCandidateRoutes();
		ELSIF cmd_bNext THEN
			machineState := TABLEMANAGER_DOOR_TRACKER_FINDPATH_FIND_SEARCH_RESULTS;
		END_IF
		
	TABLEMANAGER_DOOR_TRACKER_FINDPATH_FIND_SEARCH_RESULTS:
		IF bFirstPass THEN
			findSearchResults();
		ELSIF cmd_bNext THEN
			machineState := TABLEMANAGER_DOOR_TRACKER_FINDPATH_COMPUTE_FINAL_SCORE;
		END_IF
	
	TABLEMANAGER_DOOR_TRACKER_FINDPATH_COMPUTE_FINAL_SCORE:
		IF bFirstPass THEN
			computeFinalScore();
		ELSIF cmd_bNext THEN
			IF bFoundValidRoute THEN
				machineState := TABLEMANAGER_DOOR_TRACKER_FINDPATH_COMPLETE;
			ELSIF cmd_bNewRouteRequested THEN
				IF NOT (cmd_bNewRouteRequestedFromDoorHasNoTarget AND stDoorTrack.Target = -1) THEN
					// restore to last door track. 
					stDoorTrack := stDoorTrackLast;
				END_IF
				machineState := TABLEMANAGER_DOOR_TRACKER_FINDPATH_COMPLETE;
			ELSE				
				machineState := TABLEMANAGER_DOOR_TRACKER_FINDPATH_WAITING_FOR_CLEAR_ROUTE;
			END_IF			
		END_IF
	
	TABLEMANAGER_DOOR_TRACKER_FINDPATH_REQUEST_NEW_ROUTE_COMPLETE:
		IF bFirstPass THEN
			cmd_bRequestNewRoute := FALSE;			
		ELSE
			IF cmd_bNewRouteRequestedFromWaitingForClearRoute THEN
				machineState := TABLEMANAGER_DOOR_TRACKER_FINDPATH_WAITING_FOR_CLEAR_ROUTE;
			ELSIF cmd_bNewRouteRequestedFromAllTargetFeedoutPortsDisabled THEN
				machineState := TABLEMANAGER_DOOR_TRACKER_ALL_TARGET_FEEDOUT_PORTS_DISABLED;
			ELSIF cmd_bNewRouteRequestedFromDoorHasNoTarget THEN
				machineState := TABLEMANAGER_DOOR_TRACKER_DOOR_HAS_NO_TARGET;
			ELSIF cmd_bNewRouteRequestedFromDoorInMachineIdle OR 
				cmd_bNewRouteRequestedFromWaitForFeedout THEN
				machineState := TABLEMANAGER_DOOR_TRACKER_DOOR_IN_MACHINE_IDLE;
			ELSIF cmd_bNext THEN
				machineState := TABLEMANAGER_DOOR_TRACKER_FINDPATH_COMPLETE;				
			END_IF
			cmd_bNewRouteRequestedFromWaitingForClearRoute := FALSE;
			cmd_bNewRouteRequestedFromAllTargetFeedoutPortsDisabled := FALSE;
			cmd_bNewRouteRequestedFromDoorHasNoTarget := FALSE;
			cmd_bNewRouteRequestedFromDoorInMachineIdle := FALSE;
			cmd_bNewRouteRequestedFromWaitForFeedout := FALSE;					
		END_IF
	
	TABLEMANAGER_DOOR_TRACKER_FINDPATH_COMPLETE:
		IF bFirstPass THEN
			bFindingPath := FALSE;
			cmd_bNewTargetFeedoutPortSelected := FALSE;
			cmd_bNewRouteRequested := FALSE;	
			IF cmd_bRequestNewRoute THEN
				machineState := TABLEMANAGER_DOOR_TRACKER_FINDPATH_REQUEST_NEW_ROUTE_COMPLETE;
			ELSIF cmd_bNext THEN
				IF bHasDoor THEN
					machineState := TABLEMANAGER_DOOR_TRACKER_DOOR_IN_MACHINE_IDLE;
				ELSE
					machineState := TABLEMANAGER_DOOR_TRACKER_ROUTE_READY_WAIT_FOR_FEED_IN;
				END_IF
			END_IF
		END_IF
		
	TABLEMANAGER_DOOR_TRACKER_ALL_TARGET_FEEDOUT_PORTS_DISABLED:
		IF bFirstPass THEN
			bFindingPath := FALSE;
			cmd_bRequestNewRoute := FALSE;
			cmd_bNewTargetFeedoutPortSelected := FALSE;
			setReadyToFeedoutSides(FALSE);
		ELSE
			IF cmd_bRequestNewRoute THEN
				cmd_bNewRouteRequestedFromAllTargetFeedoutPortsDisabled:=TRUE;
				machineState := TABLEMANAGER_DOOR_TRACKER_START;
			ELSIF cmd_bNewTargetFeedoutPortSelected THEN
				machineState := TABLEMANAGER_DOOR_TRACKER_START;
			ELSIF ftrigAllTargetFeedoutPortsDisabled.Q THEN
				machineState := TABLEMANAGER_DOOR_TRACKER_START;
			ELSIF NOT cmd_bAutoFeedOn THEN
				machineState := TABLEMANAGER_AUTOFEED_OFF;
			END_IF
		END_IF
	
	TABLEMANAGER_DOOR_TRACKER_DOOR_HAS_NO_TARGET:
		IF bFirstPass THEN
			bFindingPath := FALSE;
			cmd_bRequestNewRoute := FALSE;
			cmd_bNewTargetFeedoutPortSelected := FALSE;
			setReadyToFeedoutSides(FALSE);	
			setNextDoorId();	
			initInputSourceAndDestinationIndexWithHighestFeedoutPortsCount(stDoorTrack.Source, stDoorTrack.DestinationIndex);
		ELSE
			IF cmd_bRequestNewRoute THEN
				cmd_bDoorHasNoTarget := FALSE;
				cmd_bNewRouteRequestedFromDoorHasNoTarget:=TRUE;
				machineState := TABLEMANAGER_DOOR_TRACKER_START;
			ELSIF cmd_bNewTargetFeedoutPortSelected THEN
				machineState := TABLEMANAGER_DOOR_TRACKER_START;
			ELSIF ftrigDoorHasNoTarget.Q THEN
				cmd_bDoorHasNoTarget := FALSE;
				machineState := TABLEMANAGER_DOOR_TRACKER_START;
			ELSIF NOT cmd_bAutoFeedOn THEN
				machineState := TABLEMANAGER_AUTOFEED_OFF;
			END_IF
		END_IF
		
	TABLEMANAGER_ERROR:
		IF (bFirstPass) THEN
			bError := TRUE;	
			status_bBusy := FALSE;
			cmd_bAutoFeedOn := FALSE;
			bExternal := FALSE;
		END_IF
		IF cmd_bReset THEN
			smDoorDasher.cmd_bReset := TRUE;
			smC234FeedManager.cmd_bReset := TRUE;
			smC235FeedManager.cmd_bReset := TRUE;
			clearLastError();
			machineState := TABLEMANAGER_AUTOFEED_OFF;
		END_IF




END_CASE
END_METHOD

(* The UML-statechart version of the Structured-Text version of doState method.  
	The derived function block of KvalStateMachineBase_UmlSC should override/extend this method.  *)
METHOD doState_UmlSC
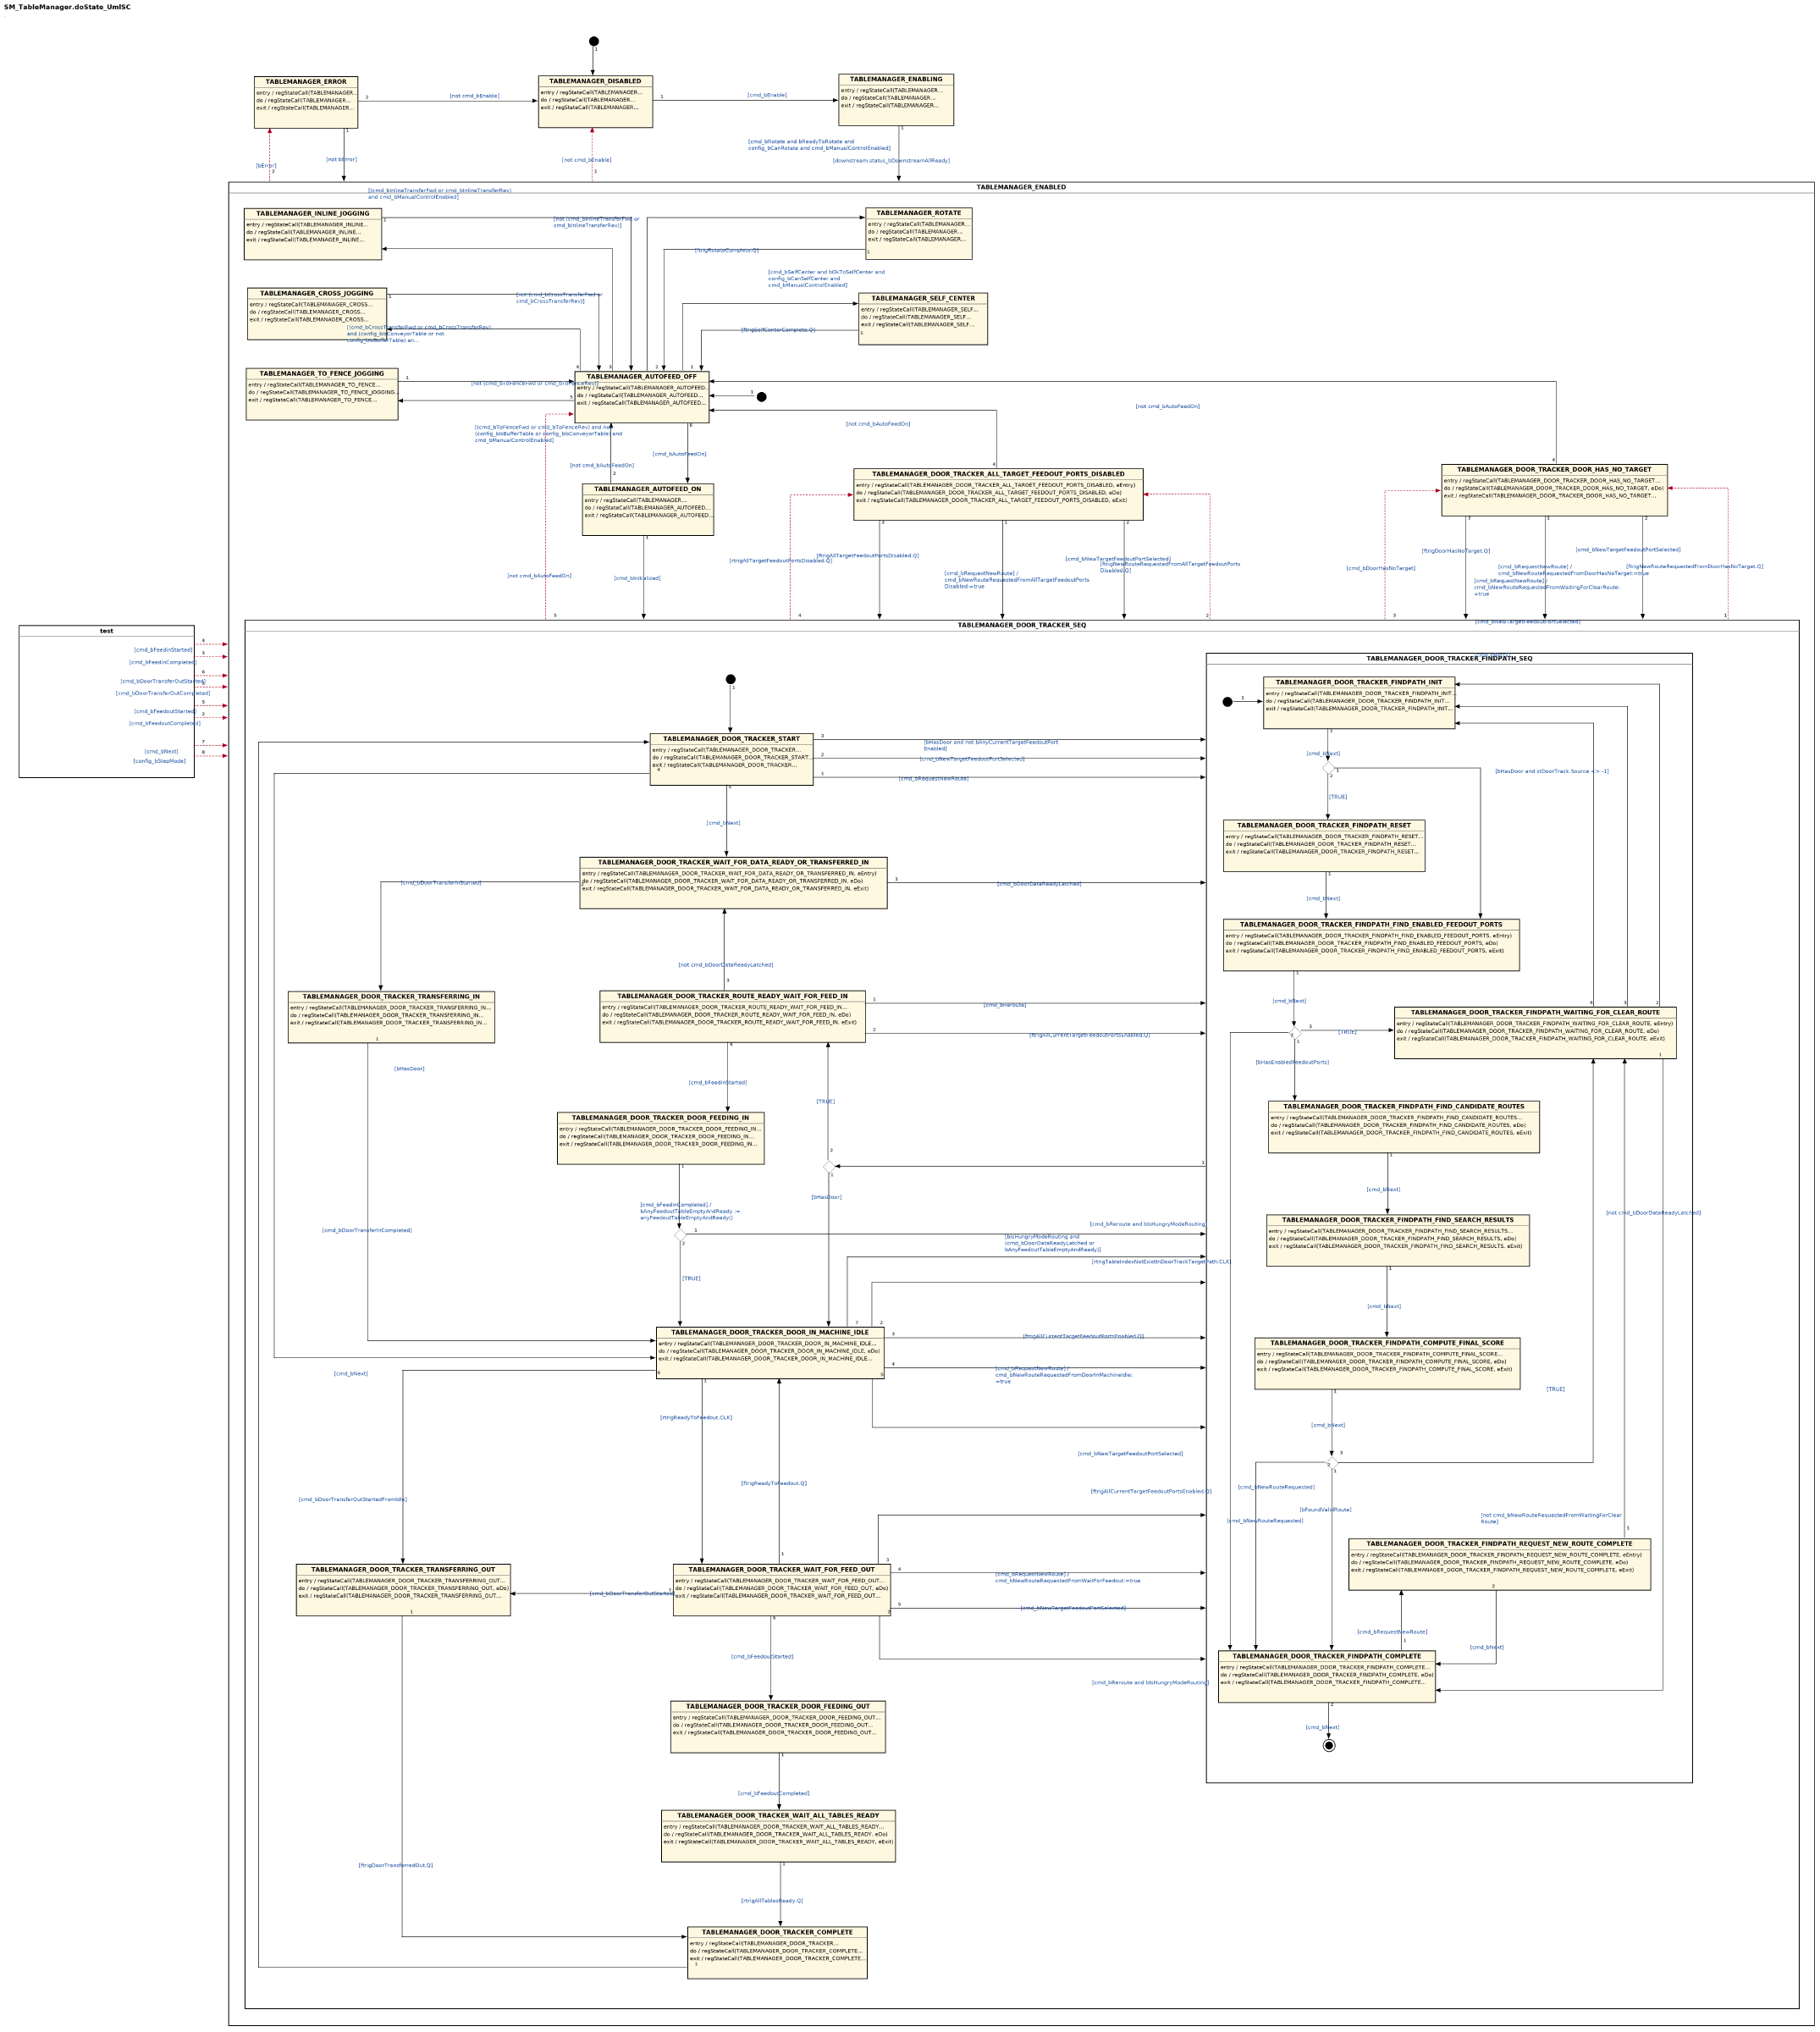
STATECHART doState_UmlSC  // abortable
    START StartState1
    STATE TABLEMANAGER_ERROR
        entry / regStateCall(TABLEMANAGER_ERROR, eEntry)
        do / regStateCall(TABLEMANAGER_ERROR, eDo)
        exit / regStateCall(TABLEMANAGER_ERROR, eExit)
    STATE TABLEMANAGER_DISABLED
        entry / regStateCall(TABLEMANAGER_DISABLED, eEntry)
        do / regStateCall(TABLEMANAGER_DISABLED, eDo)
        exit / regStateCall(TABLEMANAGER_DISABLED, eExit)
    STATE TABLEMANAGER_ENABLING
        entry / regStateCall(TABLEMANAGER_ENABLING, eEntry)
        do / regStateCall(TABLEMANAGER_ENABLING, eDo)
        exit / regStateCall(TABLEMANAGER_ENABLING, eExit)
    COMPOSITE STATE TABLEMANAGER_ENABLED
        START StartState1_copy
        NOTEELEMENT 
        STATE TABLEMANAGER_INLINE_JOGGING
            entry / regStateCall(TABLEMANAGER_INLINE_JOGGING, eEntry)
            do / regStateCall(TABLEMANAGER_INLINE_JOGGING, eDo)
            exit / regStateCall(TABLEMANAGER_INLINE_JOGGING, eExit)
        STATE TABLEMANAGER_ROTATE
            entry / regStateCall(TABLEMANAGER_ROTATE, eEntry)
            do / regStateCall(TABLEMANAGER_ROTATE, eDo)
            exit / regStateCall(TABLEMANAGER_ROTATE, eExit)
        STATE TABLEMANAGER_CROSS_JOGGING
            entry / regStateCall(TABLEMANAGER_CROSS_JOGGING, eEntry)
            do / regStateCall(TABLEMANAGER_CROSS_JOGGING, eDo)
            exit / regStateCall(TABLEMANAGER_CROSS_JOGGING, eExit)
        STATE TABLEMANAGER_SELF_CENTER
            entry / regStateCall(TABLEMANAGER_SELF_CENTER, eEntry)
            do / regStateCall(TABLEMANAGER_SELF_CENTER, eDo)
            exit / regStateCall(TABLEMANAGER_SELF_CENTER, eExit)
        STATE TABLEMANAGER_TO_FENCE_JOGGING
            entry / regStateCall(TABLEMANAGER_TO_FENCE_JOGGING, eEntry)
            do / regStateCall(TABLEMANAGER_TO_FENCE_JOGGING, eDo)
            exit / regStateCall(TABLEMANAGER_TO_FENCE_JOGGING, eExit)
        STATE TABLEMANAGER_AUTOFEED_OFF
            entry / regStateCall(TABLEMANAGER_AUTOFEED_OFF, eEntry)
            do / regStateCall(TABLEMANAGER_AUTOFEED_OFF, eDo)
            exit / regStateCall(TABLEMANAGER_AUTOFEED_OFF, eExit)
        STATE TABLEMANAGER_DOOR_TRACKER_DOOR_HAS_NO_TARGET
            entry / regStateCall(TABLEMANAGER_DOOR_TRACKER_DOOR_HAS_NO_TARGET, eEntry)
            do / regStateCall(TABLEMANAGER_DOOR_TRACKER_DOOR_HAS_NO_TARGET, eDo)
            exit / regStateCall(TABLEMANAGER_DOOR_TRACKER_DOOR_HAS_NO_TARGET, eExit)
        STATE TABLEMANAGER_AUTOFEED_ON
            entry / regStateCall(TABLEMANAGER_AUTOFEED_ON, eEntry)
            do / regStateCall(TABLEMANAGER_AUTOFEED_ON, eDo)
            exit / regStateCall(TABLEMANAGER_AUTOFEED_ON, eExit)
        STATE TABLEMANAGER_DOOR_TRACKER_ALL_TARGET_FEEDOUT_PORTS_DISABLED
            entry / regStateCall(TABLEMANAGER_DOOR_TRACKER_ALL_TARGET_FEEDOUT_PORTS_DISABLED, eEntry)
            do / regStateCall(TABLEMANAGER_DOOR_TRACKER_ALL_TARGET_FEEDOUT_PORTS_DISABLED, eDo)
            exit / regStateCall(TABLEMANAGER_DOOR_TRACKER_ALL_TARGET_FEEDOUT_PORTS_DISABLED, eExit)
        COMPOSITE STATE TABLEMANAGER_DOOR_TRACKER_SEQ
            START StartState2
            NOTEELEMENT 
            NOTEELEMENT 
            NOTEELEMENT 
            NOTEELEMENT 
            NOTEELEMENT 
            NOTEELEMENT 
            NOTEELEMENT 
            NOTEELEMENT 
            NOTEELEMENT 
            NOTEELEMENT 
            NOTEELEMENT 
            NOTEELEMENT 
            NOTEELEMENT 
            NOTEELEMENT 
            NOTEELEMENT 
            NOTEELEMENT 
            NOTEELEMENT 
            NOTEELEMENT 
            NOTEELEMENT 
            COMPOSITE STATE TABLEMANAGER_DOOR_TRACKER_FINDPATH_SEQ
                START StartState3
                STATE TABLEMANAGER_DOOR_TRACKER_FINDPATH_INIT
                    entry / regStateCall(TABLEMANAGER_DOOR_TRACKER_FINDPATH_INIT, eEntry)
                    do / regStateCall(TABLEMANAGER_DOOR_TRACKER_FINDPATH_INIT, eDo)
                    exit / regStateCall(TABLEMANAGER_DOOR_TRACKER_FINDPATH_INIT, eExit)
                CHOICE ChoiceElement4
                STATE TABLEMANAGER_DOOR_TRACKER_FINDPATH_RESET
                    entry / regStateCall(TABLEMANAGER_DOOR_TRACKER_FINDPATH_RESET, eEntry)
                    do / regStateCall(TABLEMANAGER_DOOR_TRACKER_FINDPATH_RESET, eDo)
                    exit / regStateCall(TABLEMANAGER_DOOR_TRACKER_FINDPATH_RESET, eExit)
                STATE TABLEMANAGER_DOOR_TRACKER_FINDPATH_FIND_ENABLED_FEEDOUT_PORTS
                    entry / regStateCall(TABLEMANAGER_DOOR_TRACKER_FINDPATH_FIND_ENABLED_FEEDOUT_PORTS, eEntry)
                    do / regStateCall(TABLEMANAGER_DOOR_TRACKER_FINDPATH_FIND_ENABLED_FEEDOUT_PORTS, eDo)
                    exit / regStateCall(TABLEMANAGER_DOOR_TRACKER_FINDPATH_FIND_ENABLED_FEEDOUT_PORTS, eExit)
                STATE TABLEMANAGER_DOOR_TRACKER_FINDPATH_WAITING_FOR_CLEAR_ROUTE
                    entry / regStateCall(TABLEMANAGER_DOOR_TRACKER_FINDPATH_WAITING_FOR_CLEAR_ROUTE, eEntry)
                    do / regStateCall(TABLEMANAGER_DOOR_TRACKER_FINDPATH_WAITING_FOR_CLEAR_ROUTE, eDo)
                    exit / regStateCall(TABLEMANAGER_DOOR_TRACKER_FINDPATH_WAITING_FOR_CLEAR_ROUTE, eExit)
                CHOICE ChoiceElement3
                STATE TABLEMANAGER_DOOR_TRACKER_FINDPATH_FIND_CANDIDATE_ROUTES
                    entry / regStateCall(TABLEMANAGER_DOOR_TRACKER_FINDPATH_FIND_CANDIDATE_ROUTES, eEntry)
                    do / regStateCall(TABLEMANAGER_DOOR_TRACKER_FINDPATH_FIND_CANDIDATE_ROUTES, eDo)
                    exit / regStateCall(TABLEMANAGER_DOOR_TRACKER_FINDPATH_FIND_CANDIDATE_ROUTES, eExit)
                STATE TABLEMANAGER_DOOR_TRACKER_FINDPATH_FIND_SEARCH_RESULTS
                    entry / regStateCall(TABLEMANAGER_DOOR_TRACKER_FINDPATH_FIND_SEARCH_RESULTS, eEntry)
                    do / regStateCall(TABLEMANAGER_DOOR_TRACKER_FINDPATH_FIND_SEARCH_RESULTS, eDo)
                    exit / regStateCall(TABLEMANAGER_DOOR_TRACKER_FINDPATH_FIND_SEARCH_RESULTS, eExit)
                STATE TABLEMANAGER_DOOR_TRACKER_FINDPATH_COMPUTE_FINAL_SCORE
                    entry / regStateCall(TABLEMANAGER_DOOR_TRACKER_FINDPATH_COMPUTE_FINAL_SCORE, eEntry)
                    do / regStateCall(TABLEMANAGER_DOOR_TRACKER_FINDPATH_COMPUTE_FINAL_SCORE, eDo)
                    exit / regStateCall(TABLEMANAGER_DOOR_TRACKER_FINDPATH_COMPUTE_FINAL_SCORE, eExit)
                CHOICE ChoiceElement2
                STATE TABLEMANAGER_DOOR_TRACKER_FINDPATH_REQUEST_NEW_ROUTE_COMPLETE
                    entry / regStateCall(TABLEMANAGER_DOOR_TRACKER_FINDPATH_REQUEST_NEW_ROUTE_COMPLETE, eEntry)
                    do / regStateCall(TABLEMANAGER_DOOR_TRACKER_FINDPATH_REQUEST_NEW_ROUTE_COMPLETE, eDo)
                    exit / regStateCall(TABLEMANAGER_DOOR_TRACKER_FINDPATH_REQUEST_NEW_ROUTE_COMPLETE, eExit)
                STATE TABLEMANAGER_DOOR_TRACKER_FINDPATH_COMPLETE
                    entry / regStateCall(TABLEMANAGER_DOOR_TRACKER_FINDPATH_COMPLETE, eEntry)
                    do / regStateCall(TABLEMANAGER_DOOR_TRACKER_FINDPATH_COMPLETE, eDo)
                    exit / regStateCall(TABLEMANAGER_DOOR_TRACKER_FINDPATH_COMPLETE, eExit)
                END EndState2
                StartState3 -> TABLEMANAGER_DOOR_TRACKER_FINDPATH_INIT  // priority 1, on completion
                TABLEMANAGER_DOOR_TRACKER_FINDPATH_INIT -> ChoiceElement4 [cmd_bNext] // priority 1
                ChoiceElement4 -> TABLEMANAGER_DOOR_TRACKER_FINDPATH_FIND_ENABLED_FEEDOUT_PORTS [bHasDoor and stDoorTrack.Source <> -1] // priority 1
                ChoiceElement4 -> TABLEMANAGER_DOOR_TRACKER_FINDPATH_RESET [TRUE] // priority 2
                TABLEMANAGER_DOOR_TRACKER_FINDPATH_RESET -> TABLEMANAGER_DOOR_TRACKER_FINDPATH_FIND_ENABLED_FEEDOUT_PORTS [cmd_bNext] // priority 1
                TABLEMANAGER_DOOR_TRACKER_FINDPATH_FIND_ENABLED_FEEDOUT_PORTS -> ChoiceElement3 [cmd_bNext] // priority 1
                TABLEMANAGER_DOOR_TRACKER_FINDPATH_WAITING_FOR_CLEAR_ROUTE -> TABLEMANAGER_DOOR_TRACKER_FINDPATH_COMPLETE [not cmd_bDoorDataReadyLatched] // priority 1, rising edge
                TABLEMANAGER_DOOR_TRACKER_FINDPATH_WAITING_FOR_CLEAR_ROUTE -> TABLEMANAGER_DOOR_TRACKER_FINDPATH_INIT [cmd_bRequestNewRoute] / cmd_bNewRouteRequestedFromWaitingForClearRoute:=true // priority 2, rising edge
                TABLEMANAGER_DOOR_TRACKER_FINDPATH_WAITING_FOR_CLEAR_ROUTE -> TABLEMANAGER_DOOR_TRACKER_FINDPATH_INIT [cmd_bNewTargetFeedoutPortSelected] // priority 3, rising edge
                TABLEMANAGER_DOOR_TRACKER_FINDPATH_WAITING_FOR_CLEAR_ROUTE -> TABLEMANAGER_DOOR_TRACKER_FINDPATH_INIT [cmd_bRetry] // priority 4, rising edge
                ChoiceElement3 -> TABLEMANAGER_DOOR_TRACKER_FINDPATH_FIND_CANDIDATE_ROUTES [bHasEnabledFeedoutPorts] // priority 1
                ChoiceElement3 -> TABLEMANAGER_DOOR_TRACKER_FINDPATH_COMPLETE [cmd_bNewRouteRequested] // priority 2
                ChoiceElement3 -> TABLEMANAGER_DOOR_TRACKER_FINDPATH_WAITING_FOR_CLEAR_ROUTE [TRUE] // priority 3
                TABLEMANAGER_DOOR_TRACKER_FINDPATH_FIND_CANDIDATE_ROUTES -> TABLEMANAGER_DOOR_TRACKER_FINDPATH_FIND_SEARCH_RESULTS [cmd_bNext] // priority 1
                TABLEMANAGER_DOOR_TRACKER_FINDPATH_FIND_SEARCH_RESULTS -> TABLEMANAGER_DOOR_TRACKER_FINDPATH_COMPUTE_FINAL_SCORE [cmd_bNext] // priority 1
                TABLEMANAGER_DOOR_TRACKER_FINDPATH_COMPUTE_FINAL_SCORE -> ChoiceElement2 [cmd_bNext] // priority 1
                ChoiceElement2 -> TABLEMANAGER_DOOR_TRACKER_FINDPATH_COMPLETE [bFoundValidRoute] // priority 1
                ChoiceElement2 -> TABLEMANAGER_DOOR_TRACKER_FINDPATH_COMPLETE [cmd_bNewRouteRequested] // priority 2
                ChoiceElement2 -> TABLEMANAGER_DOOR_TRACKER_FINDPATH_WAITING_FOR_CLEAR_ROUTE [TRUE] // priority 3
                TABLEMANAGER_DOOR_TRACKER_FINDPATH_REQUEST_NEW_ROUTE_COMPLETE -> TABLEMANAGER_DOOR_TRACKER_FINDPATH_WAITING_FOR_CLEAR_ROUTE [not cmd_bNewRouteRequestedFromWaitingForClearRoute] // priority 1, rising edge
                TABLEMANAGER_DOOR_TRACKER_FINDPATH_REQUEST_NEW_ROUTE_COMPLETE -> TABLEMANAGER_DOOR_TRACKER_FINDPATH_COMPLETE [cmd_bNext] // priority 2
                TABLEMANAGER_DOOR_TRACKER_FINDPATH_COMPLETE -> TABLEMANAGER_DOOR_TRACKER_FINDPATH_REQUEST_NEW_ROUTE_COMPLETE [cmd_bRequestNewRoute] // priority 1
                TABLEMANAGER_DOOR_TRACKER_FINDPATH_COMPLETE -> EndState2 [cmd_bNext] // priority 2
            END_STATE
            STATE TABLEMANAGER_DOOR_TRACKER_START
                entry / regStateCall(TABLEMANAGER_DOOR_TRACKER_START, eEntry)
                do / regStateCall(TABLEMANAGER_DOOR_TRACKER_START, eDo)
                exit / regStateCall(TABLEMANAGER_DOOR_TRACKER_START, eExit)
            STATE TABLEMANAGER_DOOR_TRACKER_WAIT_FOR_DATA_READY_OR_TRANSFERRED_IN
                entry / regStateCall(TABLEMANAGER_DOOR_TRACKER_WAIT_FOR_DATA_READY_OR_TRANSFERRED_IN, eEntry)
                do / regStateCall(TABLEMANAGER_DOOR_TRACKER_WAIT_FOR_DATA_READY_OR_TRANSFERRED_IN, eDo)
                exit / regStateCall(TABLEMANAGER_DOOR_TRACKER_WAIT_FOR_DATA_READY_OR_TRANSFERRED_IN, eExit)
            STATE TABLEMANAGER_DOOR_TRACKER_TRANSFERRING_IN
                entry / regStateCall(TABLEMANAGER_DOOR_TRACKER_TRANSFERRING_IN, eEntry)
                do / regStateCall(TABLEMANAGER_DOOR_TRACKER_TRANSFERRING_IN, eDo)
                exit / regStateCall(TABLEMANAGER_DOOR_TRACKER_TRANSFERRING_IN, eExit)
            STATE TABLEMANAGER_DOOR_TRACKER_ROUTE_READY_WAIT_FOR_FEED_IN
                entry / regStateCall(TABLEMANAGER_DOOR_TRACKER_ROUTE_READY_WAIT_FOR_FEED_IN, eEntry)
                do / regStateCall(TABLEMANAGER_DOOR_TRACKER_ROUTE_READY_WAIT_FOR_FEED_IN, eDo)
                exit / regStateCall(TABLEMANAGER_DOOR_TRACKER_ROUTE_READY_WAIT_FOR_FEED_IN, eExit)
            STATE TABLEMANAGER_DOOR_TRACKER_DOOR_FEEDING_IN
                entry / regStateCall(TABLEMANAGER_DOOR_TRACKER_DOOR_FEEDING_IN, eEntry)
                do / regStateCall(TABLEMANAGER_DOOR_TRACKER_DOOR_FEEDING_IN, eDo)
                exit / regStateCall(TABLEMANAGER_DOOR_TRACKER_DOOR_FEEDING_IN, eExit)
            CHOICE ChoiceElement1
            CHOICE ChoiceElement5
            STATE TABLEMANAGER_DOOR_TRACKER_DOOR_IN_MACHINE_IDLE
                entry / regStateCall(TABLEMANAGER_DOOR_TRACKER_DOOR_IN_MACHINE_IDLE, eEntry)
                do / regStateCall(TABLEMANAGER_DOOR_TRACKER_DOOR_IN_MACHINE_IDLE, eDo)
                exit / regStateCall(TABLEMANAGER_DOOR_TRACKER_DOOR_IN_MACHINE_IDLE, eExit)
            STATE TABLEMANAGER_DOOR_TRACKER_TRANSFERRING_OUT
                entry / regStateCall(TABLEMANAGER_DOOR_TRACKER_TRANSFERRING_OUT, eEntry)
                do / regStateCall(TABLEMANAGER_DOOR_TRACKER_TRANSFERRING_OUT, eDo)
                exit / regStateCall(TABLEMANAGER_DOOR_TRACKER_TRANSFERRING_OUT, eExit)
            STATE TABLEMANAGER_DOOR_TRACKER_WAIT_FOR_FEED_OUT
                entry / regStateCall(TABLEMANAGER_DOOR_TRACKER_WAIT_FOR_FEED_OUT, eEntry)
                do / regStateCall(TABLEMANAGER_DOOR_TRACKER_WAIT_FOR_FEED_OUT, eDo)
                exit / regStateCall(TABLEMANAGER_DOOR_TRACKER_WAIT_FOR_FEED_OUT, eExit)
            STATE TABLEMANAGER_DOOR_TRACKER_DOOR_FEEDING_OUT
                entry / regStateCall(TABLEMANAGER_DOOR_TRACKER_DOOR_FEEDING_OUT, eEntry)
                do / regStateCall(TABLEMANAGER_DOOR_TRACKER_DOOR_FEEDING_OUT, eDo)
                exit / regStateCall(TABLEMANAGER_DOOR_TRACKER_DOOR_FEEDING_OUT, eExit)
            STATE TABLEMANAGER_DOOR_TRACKER_WAIT_ALL_TABLES_READY
                entry / regStateCall(TABLEMANAGER_DOOR_TRACKER_WAIT_ALL_TABLES_READY, eEntry)
                do / regStateCall(TABLEMANAGER_DOOR_TRACKER_WAIT_ALL_TABLES_READY, eDo)
                exit / regStateCall(TABLEMANAGER_DOOR_TRACKER_WAIT_ALL_TABLES_READY, eExit)
            STATE TABLEMANAGER_DOOR_TRACKER_COMPLETE
                entry / regStateCall(TABLEMANAGER_DOOR_TRACKER_COMPLETE, eEntry)
                do / regStateCall(TABLEMANAGER_DOOR_TRACKER_COMPLETE, eDo)
                exit / regStateCall(TABLEMANAGER_DOOR_TRACKER_COMPLETE, eExit)
            StartState2 -> TABLEMANAGER_DOOR_TRACKER_START  // priority 1, on completion
            TABLEMANAGER_DOOR_TRACKER_FINDPATH_SEQ -> ChoiceElement1  // priority 1, on completion
            TABLEMANAGER_DOOR_TRACKER_START -> TABLEMANAGER_DOOR_TRACKER_FINDPATH_SEQ [cmd_bRequestNewRoute] // priority 1
            TABLEMANAGER_DOOR_TRACKER_START -> TABLEMANAGER_DOOR_TRACKER_FINDPATH_SEQ [cmd_bNewTargetFeedoutPortSelected] // priority 2
            TABLEMANAGER_DOOR_TRACKER_START -> TABLEMANAGER_DOOR_TRACKER_FINDPATH_SEQ [bHasDoor and not bAnyCurrentTargetFeedoutPortEnabled] // priority 3
            TABLEMANAGER_DOOR_TRACKER_START -> TABLEMANAGER_DOOR_TRACKER_DOOR_IN_MACHINE_IDLE [bHasDoor] // priority 4
            TABLEMANAGER_DOOR_TRACKER_START -> TABLEMANAGER_DOOR_TRACKER_WAIT_FOR_DATA_READY_OR_TRANSFERRED_IN [cmd_bNext] // priority 5
            TABLEMANAGER_DOOR_TRACKER_WAIT_FOR_DATA_READY_OR_TRANSFERRED_IN -> TABLEMANAGER_DOOR_TRACKER_FINDPATH_SEQ [cmd_bDoorDataReadyLatched] // priority 1
            TABLEMANAGER_DOOR_TRACKER_WAIT_FOR_DATA_READY_OR_TRANSFERRED_IN -> TABLEMANAGER_DOOR_TRACKER_TRANSFERRING_IN [cmd_bDoorTransferInStarted] // priority 2, rising edge
            TABLEMANAGER_DOOR_TRACKER_TRANSFERRING_IN -> TABLEMANAGER_DOOR_TRACKER_DOOR_IN_MACHINE_IDLE [cmd_bDoorTransferInCompleted] // priority 1, rising edge
            TABLEMANAGER_DOOR_TRACKER_ROUTE_READY_WAIT_FOR_FEED_IN -> TABLEMANAGER_DOOR_TRACKER_FINDPATH_SEQ [cmd_bReroute] // priority 1
            TABLEMANAGER_DOOR_TRACKER_ROUTE_READY_WAIT_FOR_FEED_IN -> TABLEMANAGER_DOOR_TRACKER_FINDPATH_SEQ [ftrigAllCurrentTargetFeedoutPortsEnabled.Q] // priority 2, rising edge
            TABLEMANAGER_DOOR_TRACKER_ROUTE_READY_WAIT_FOR_FEED_IN -> TABLEMANAGER_DOOR_TRACKER_WAIT_FOR_DATA_READY_OR_TRANSFERRED_IN [not cmd_bDoorDataReadyLatched] // priority 3
            TABLEMANAGER_DOOR_TRACKER_ROUTE_READY_WAIT_FOR_FEED_IN -> TABLEMANAGER_DOOR_TRACKER_DOOR_FEEDING_IN [cmd_bFeedinStarted] // priority 4, rising edge
            TABLEMANAGER_DOOR_TRACKER_DOOR_FEEDING_IN -> ChoiceElement5 [cmd_bFeedinCompleted] / bAnyFeedoutTableEmptyAndReady := anyFeedoutTableEmptyAndReady() // priority 1, rising edge
            ChoiceElement1 -> TABLEMANAGER_DOOR_TRACKER_DOOR_IN_MACHINE_IDLE [bHasDoor] // priority 1
            ChoiceElement1 -> TABLEMANAGER_DOOR_TRACKER_ROUTE_READY_WAIT_FOR_FEED_IN [TRUE] // priority 2
            ChoiceElement5 -> TABLEMANAGER_DOOR_TRACKER_FINDPATH_SEQ [bIsHungryModeRouting and (cmd_bDoorDataReadyLatched or bAnyFeedoutTableEmptyAndReady)] // priority 1
            ChoiceElement5 -> TABLEMANAGER_DOOR_TRACKER_DOOR_IN_MACHINE_IDLE [TRUE] // priority 2
            TABLEMANAGER_DOOR_TRACKER_DOOR_IN_MACHINE_IDLE -> TABLEMANAGER_DOOR_TRACKER_WAIT_FOR_FEED_OUT [rtrigReadyToFeedout.CLK] // priority 1
            TABLEMANAGER_DOOR_TRACKER_DOOR_IN_MACHINE_IDLE -> TABLEMANAGER_DOOR_TRACKER_FINDPATH_SEQ [rtrigTableIndexNotExistInDoorTrackTargetPath.CLK] // priority 2
            TABLEMANAGER_DOOR_TRACKER_DOOR_IN_MACHINE_IDLE -> TABLEMANAGER_DOOR_TRACKER_FINDPATH_SEQ [ftrigAllCurrentTargetFeedoutPortsEnabled.Q] // priority 3, rising edge
            TABLEMANAGER_DOOR_TRACKER_DOOR_IN_MACHINE_IDLE -> TABLEMANAGER_DOOR_TRACKER_FINDPATH_SEQ [cmd_bRequestNewRoute] / cmd_bNewRouteRequestedFromDoorInMachineIdle:=true // priority 4, rising edge
            TABLEMANAGER_DOOR_TRACKER_DOOR_IN_MACHINE_IDLE -> TABLEMANAGER_DOOR_TRACKER_FINDPATH_SEQ [cmd_bNewTargetFeedoutPortSelected] // priority 5, rising edge
            TABLEMANAGER_DOOR_TRACKER_DOOR_IN_MACHINE_IDLE -> TABLEMANAGER_DOOR_TRACKER_TRANSFERRING_OUT [cmd_bDoorTransferOutStartedFromIdle] // priority 6
            TABLEMANAGER_DOOR_TRACKER_DOOR_IN_MACHINE_IDLE -> TABLEMANAGER_DOOR_TRACKER_FINDPATH_SEQ [cmd_bReroute and bIsHungryModeRouting] // priority 7
            TABLEMANAGER_DOOR_TRACKER_TRANSFERRING_OUT -> TABLEMANAGER_DOOR_TRACKER_COMPLETE [ftrigDoorTransferredOut.Q] // priority 1, rising edge
            TABLEMANAGER_DOOR_TRACKER_WAIT_FOR_FEED_OUT -> TABLEMANAGER_DOOR_TRACKER_DOOR_IN_MACHINE_IDLE [ftrigReadyToFeedout.Q] // priority 1, rising edge
            TABLEMANAGER_DOOR_TRACKER_WAIT_FOR_FEED_OUT -> TABLEMANAGER_DOOR_TRACKER_FINDPATH_SEQ [cmd_bReroute and bIsHungryModeRouting] // priority 2
            TABLEMANAGER_DOOR_TRACKER_WAIT_FOR_FEED_OUT -> TABLEMANAGER_DOOR_TRACKER_FINDPATH_SEQ [ftrigAllCurrentTargetFeedoutPortsEnabled.Q] // priority 3, rising edge
            TABLEMANAGER_DOOR_TRACKER_WAIT_FOR_FEED_OUT -> TABLEMANAGER_DOOR_TRACKER_FINDPATH_SEQ [cmd_bRequestNewRoute] / cmd_bNewRouteRequestedFromWaitForFeedout:=true // priority 4, rising edge
            TABLEMANAGER_DOOR_TRACKER_WAIT_FOR_FEED_OUT -> TABLEMANAGER_DOOR_TRACKER_FINDPATH_SEQ [cmd_bNewTargetFeedoutPortSelected] // priority 5, rising edge
            TABLEMANAGER_DOOR_TRACKER_WAIT_FOR_FEED_OUT -> TABLEMANAGER_DOOR_TRACKER_DOOR_FEEDING_OUT [cmd_bFeedoutStarted] // priority 6, rising edge
            TABLEMANAGER_DOOR_TRACKER_WAIT_FOR_FEED_OUT -> TABLEMANAGER_DOOR_TRACKER_TRANSFERRING_OUT [cmd_bDoorTransferOutStarted] // priority 7
            TABLEMANAGER_DOOR_TRACKER_DOOR_FEEDING_OUT -> TABLEMANAGER_DOOR_TRACKER_WAIT_ALL_TABLES_READY [cmd_bFeedoutCompleted] // priority 1, rising edge
            TABLEMANAGER_DOOR_TRACKER_WAIT_ALL_TABLES_READY -> TABLEMANAGER_DOOR_TRACKER_COMPLETE [rtrigAllTablesReady.Q] // priority 1, rising edge
            TABLEMANAGER_DOOR_TRACKER_COMPLETE -> TABLEMANAGER_DOOR_TRACKER_START [cmd_bNext] // priority 1
        END_STATE
        StartState1_copy -> TABLEMANAGER_AUTOFEED_OFF  // priority 1, on completion
        TABLEMANAGER_INLINE_JOGGING -> TABLEMANAGER_AUTOFEED_OFF [not (cmd_bInlineTransferFwd or cmd_bInlineTransferRev)] // priority 1
        TABLEMANAGER_ROTATE -> TABLEMANAGER_AUTOFEED_OFF [ftrigRotateComplete.Q] // priority 1, rising edge
        TABLEMANAGER_CROSS_JOGGING -> TABLEMANAGER_AUTOFEED_OFF [not (cmd_bCrossTransferFwd or cmd_bCrossTransferRev)] // priority 1
        TABLEMANAGER_SELF_CENTER -> TABLEMANAGER_AUTOFEED_OFF [ftrigSelfCenterComplete.Q] // priority 1, rising edge
        TABLEMANAGER_TO_FENCE_JOGGING -> TABLEMANAGER_AUTOFEED_OFF [not (cmd_bToFenceFwd or cmd_bToFenceRev)] // priority 1
        TABLEMANAGER_AUTOFEED_OFF -> TABLEMANAGER_SELF_CENTER [cmd_bSelfCenter and bOkToSelfCenter and config_bCanSelfCenter and cmd_bManualControlEnabled] // priority 1, rising edge
        TABLEMANAGER_AUTOFEED_OFF -> TABLEMANAGER_ROTATE [cmd_bRotate and bReadyToRotate and config_bCanRotate and cmd_bManualControlEnabled] // priority 2, rising edge
        TABLEMANAGER_AUTOFEED_OFF -> TABLEMANAGER_INLINE_JOGGING [(cmd_bInlineTransferFwd or cmd_bInlineTransferRev) and cmd_bManualControlEnabled] // priority 3
        TABLEMANAGER_AUTOFEED_OFF -> TABLEMANAGER_CROSS_JOGGING [(cmd_bCrossTransferFwd or cmd_bCrossTransferRev) and (config_bIsConveyorTable or not config_bIsBufferTable) and cmd_bManualControlEnabled] // priority 4
        TABLEMANAGER_AUTOFEED_OFF -> TABLEMANAGER_TO_FENCE_JOGGING [(cmd_bToFenceFwd or cmd_bToFenceRev) and not (config_bIsBufferTable or config_bIsConveyorTable) and cmd_bManualControlEnabled] // priority 5
        TABLEMANAGER_AUTOFEED_OFF -> TABLEMANAGER_AUTOFEED_ON [cmd_bAutoFeedOn] // priority 6
        TABLEMANAGER_DOOR_TRACKER_DOOR_HAS_NO_TARGET -> TABLEMANAGER_DOOR_TRACKER_SEQ [cmd_bRequestNewRoute] / cmd_bNewRouteRequestedFromDoorHasNoTarget:=true // priority 1, rising edge
        TABLEMANAGER_DOOR_TRACKER_DOOR_HAS_NO_TARGET -> TABLEMANAGER_DOOR_TRACKER_SEQ [cmd_bNewTargetFeedoutPortSelected] // priority 2, rising edge
        TABLEMANAGER_DOOR_TRACKER_DOOR_HAS_NO_TARGET -> TABLEMANAGER_DOOR_TRACKER_SEQ [ftrigDoorHasNoTarget.Q] // priority 3, rising edge
        TABLEMANAGER_DOOR_TRACKER_DOOR_HAS_NO_TARGET -> TABLEMANAGER_AUTOFEED_OFF [not cmd_bAutoFeedOn] // priority 4
        TABLEMANAGER_AUTOFEED_ON -> TABLEMANAGER_DOOR_TRACKER_SEQ [cmd_bInitialized] // priority 1
        TABLEMANAGER_AUTOFEED_ON -> TABLEMANAGER_AUTOFEED_OFF [not cmd_bAutoFeedOn] // priority 2
        TABLEMANAGER_DOOR_TRACKER_ALL_TARGET_FEEDOUT_PORTS_DISABLED -> TABLEMANAGER_DOOR_TRACKER_SEQ [cmd_bRequestNewRoute] / cmd_bNewRouteRequestedFromAllTargetFeedoutPortsDisabled:=true // priority 1, rising edge
        TABLEMANAGER_DOOR_TRACKER_ALL_TARGET_FEEDOUT_PORTS_DISABLED -> TABLEMANAGER_DOOR_TRACKER_SEQ [cmd_bNewTargetFeedoutPortSelected] // priority 2, rising edge
        TABLEMANAGER_DOOR_TRACKER_ALL_TARGET_FEEDOUT_PORTS_DISABLED -> TABLEMANAGER_DOOR_TRACKER_SEQ [ftrigAllTargetFeedoutPortsDisabled.Q] // priority 3, rising edge
        TABLEMANAGER_DOOR_TRACKER_ALL_TARGET_FEEDOUT_PORTS_DISABLED -> TABLEMANAGER_AUTOFEED_OFF [not cmd_bAutoFeedOn] // priority 4
        TABLEMANAGER_DOOR_TRACKER_SEQ -> TABLEMANAGER_DOOR_TRACKER_DOOR_HAS_NO_TARGET [ftrigNewRouteRequestedFromDoorHasNoTarget.Q] // priority 1, exception, rising edge
        TABLEMANAGER_DOOR_TRACKER_SEQ -> TABLEMANAGER_DOOR_TRACKER_ALL_TARGET_FEEDOUT_PORTS_DISABLED [ftrigNewRouteRequestedFromAllTargetFeedoutPortsDisabled.Q] // priority 2, exception, rising edge
        TABLEMANAGER_DOOR_TRACKER_SEQ -> TABLEMANAGER_DOOR_TRACKER_DOOR_HAS_NO_TARGET [cmd_bDoorHasNoTarget] // priority 3, exception
        TABLEMANAGER_DOOR_TRACKER_SEQ -> TABLEMANAGER_DOOR_TRACKER_ALL_TARGET_FEEDOUT_PORTS_DISABLED [rtrigAllTargetFeedoutPortsDisabled.Q] // priority 4, exception, rising edge
        TABLEMANAGER_DOOR_TRACKER_SEQ -> TABLEMANAGER_AUTOFEED_OFF [not cmd_bAutoFeedOn] // priority 5, exception
    END_STATE
    COMPOSITE STATE test
    END_STATE
    StartState1 -> TABLEMANAGER_DISABLED  // priority 1, on completion
    TABLEMANAGER_ERROR -> TABLEMANAGER_ENABLED [not bError] // priority 1
    TABLEMANAGER_ERROR -> TABLEMANAGER_DISABLED [not cmd_bEnable] // priority 2
    TABLEMANAGER_DISABLED -> TABLEMANAGER_ENABLING [cmd_bEnable] // priority 1
    TABLEMANAGER_ENABLING -> TABLEMANAGER_ENABLED [downstream.status_bDownstreamAllReady] // priority 1
    TABLEMANAGER_ENABLED -> TABLEMANAGER_DISABLED [not cmd_bEnable] // priority 1, exception
    TABLEMANAGER_ENABLED -> TABLEMANAGER_ERROR [bError] // priority 2, exception
    test -> TABLEMANAGER_ENABLED [cmd_bDoorTransferOutCompleted] // priority 1, exception
    test -> TABLEMANAGER_ENABLED [cmd_bFeedoutCompleted] // priority 2, exception
    test -> TABLEMANAGER_ENABLED [cmd_bFeedinCompleted] // priority 3, exception
    test -> TABLEMANAGER_ENABLED [cmd_bFeedinStarted] // priority 4, exception
    test -> TABLEMANAGER_ENABLED [cmd_bFeedoutStarted] // priority 5, exception
    test -> TABLEMANAGER_ENABLED [cmd_bDoorTransferOutStarted] // priority 6, exception
    test -> TABLEMANAGER_ENABLED [cmd_bNext] // priority 7, exception
    test -> TABLEMANAGER_ENABLED [config_bStepMode] // priority 8, exception
    NOTEELEMENT 
END_STATECHART
END_METHOD

METHOD existTableIndexInDoorTrackTargetPath : BOOL
VAR
	i : INT;
	pstPath : POINTER TO ST_PathInfo;
END_VAR
existTableIndexInDoorTrackTargetPath := FALSE;

pstPath := ADR(stDoorTrack.TargetPath);

FOR i:= 0 TO pstPath^.PathCount - 1 DO
	IF pstPath^.Path[i].TableIndex = config_iTableArrayIndex THEN
		existTableIndexInDoorTrackTargetPath := TRUE;
		EXIT;
	END_IF
END_FOR
END_METHOD

METHOD findAllCandidateRoutes
VAR_INPUT
END_VAR
VAR
	i : INT;
	pstRoute : POINTER TO ST_Route; 
END_VAR
IF cmd_bRequestNewRoute THEN
	FOR i:=0 TO stDoorTrack.AllEnabledFeedoutPorts.FeedoutPortsCount - 1 DO
		pstRoute := findCandidateRoute(config_iTableArrayIndex, stDoorTrack.AllEnabledFeedoutPorts.FeedoutPorts[i].TableIndex);	
		addCandidateRouteToDoorTrack(pstRoute, stDoorTrack.AllEnabledFeedoutPorts.FeedoutPorts[i].Side);
	END_FOR
ELSE
	FOR i:=0 TO stDoorTrack.TargetFeedoutPorts.FeedoutPortsCount - 1 DO
		pstRoute := findCandidateRoute(config_iTableArrayIndex, stDoorTrack.TargetFeedoutPorts.FeedoutPorts[i].TableIndex);	
		addCandidateRouteToDoorTrack(pstRoute, stDoorTrack.TargetFeedoutPorts.FeedoutPorts[i].Side);
	END_FOR
END_IF
END_METHOD

// find all the enabled feed-out ports that are mapped to the selected DestinationIndex.
// The route planner will select the shortest path from this list in later stage.
METHOD findAllEnabledFeedoutPorts : BOOL
VAR_INPUT
END_VAR
VAR
	i : INT;
	j : INT;
	k : INT;
	stFeedoutPort : ST_FeedoutPort;
END_VAR
findAllEnabledFeedoutPorts := FALSE;
IF  stDoorTrack.DestinationIndex <> -1 AND
	stDoorTrack.Source <> -1
	THEN
	
	IF cmd_bRequestNewRoute THEN
		FOR i:=0 TO MAIN.mainStateMachine.smCtrlInterface.config_stTransferTableConfig.PrimaryTable.FeedoutPortsConfig.FeedoutPortsCount - 1 DO
			stFeedoutPort := MAIN.mainStateMachine.smCtrlInterface.config_stTransferTableConfig.PrimaryTable.FeedoutPortsConfig.FeedoutPorts[i];
			IF stDoorTrack.Target <> -1 AND stDoorTrack.Target = stFeedoutPort.TableIndex AND stDoorTrack.TargetFeedoutSide = stFeedoutPort.Side THEN
				CONTINUE;
			END_IF
			IF MAIN.mainStateMachine.asmTableManagers[stFeedoutPort.TableIndex].isFeedoutSideEnabled(stFeedoutPort.Side) THEN
				addToAllEnabledFeedoutPorts(stFeedoutPort);
			END_IF
		END_FOR
		findAllEnabledFeedoutPorts := stDoorTrack.AllEnabledFeedoutPorts.FeedoutPortsCount > 0;
	ELSIF cmd_bNewTargetFeedoutPortSelected THEN
		IF MAIN.mainStateMachine.asmTableManagers[cmd_stNewTargetFeedoutPort.TableIndex].isFeedoutSideEnabled(cmd_stNewTargetFeedoutPort.Side) THEN
			addToTargetFeedoutPorts(cmd_stNewTargetFeedoutPort);
		END_IF
		findAllEnabledFeedoutPorts := stDoorTrack.TargetFeedoutPorts.FeedoutPortsCount > 0;
	ELSIF NOT isCurrentTargetFeedoutPortExistInDestinationIndexFeedoutPorts() AND isCurrentTargetFeedoutPortEnabled() THEN
		// the current Target was a re-route, its Target's feed-out side was disabled and then re-enabled.
		stFeedoutPort.TableIndex := stDoorTrack.Target;
		stFeedoutPort.Side := stDoorTrack.TargetFeedoutSide;
		addToTargetFeedoutPorts(stFeedoutPort);
		findAllEnabledFeedoutPorts := stDoorTrack.TargetFeedoutPorts.FeedoutPortsCount > 0; 
	ELSE
		// new door wants to come in or all of Target's feed-out ports were disabled.
		i := stDoorTrack.Source;
		IF MAIN.mainStateMachine.smCtrlInterface.config_stTransferTableConfig.PrimaryTable.Tables[i].DestinationsFeedoutPortsMappingConfig.DestinationsFeedoutPortsMappingsCount > 0 THEN
			FOR j:=0 TO MAIN.mainStateMachine.smCtrlInterface.config_stTransferTableConfig.PrimaryTable.Tables[i].DestinationsFeedoutPortsMappingConfig.DestinationsFeedoutPortsMappingsCount - 1 DO
				IF MAIN.mainStateMachine.smCtrlInterface.config_stTransferTableConfig.PrimaryTable.Tables[i].DestinationsFeedoutPortsMappingConfig.DestinationsFeedoutPortsMappings[j].DestinationIndex = stDoorTrack.DestinationIndex THEN
					IF MAIN.mainStateMachine.smCtrlInterface.config_stTransferTableConfig.PrimaryTable.Tables[i].DestinationsFeedoutPortsMappingConfig.DestinationsFeedoutPortsMappings[j].FeedoutPortsCount > 0 THEN
						FOR k:=0 TO MAIN.mainStateMachine.smCtrlInterface.config_stTransferTableConfig.PrimaryTable.Tables[i].DestinationsFeedoutPortsMappingConfig.DestinationsFeedoutPortsMappings[j].FeedoutPortsCount - 1 DO
							stFeedoutPort := MAIN.mainStateMachine.smCtrlInterface.config_stTransferTableConfig.PrimaryTable.Tables[i].DestinationsFeedoutPortsMappingConfig.DestinationsFeedoutPortsMappings[j].FeedoutPorts[k];
							IF cmd_bNewRouteRequested AND stDoorTrackLast.Target = stFeedoutPort.TableIndex THEN
								CONTINUE;
							END_IF
							IF MAIN.mainStateMachine.asmTableManagers[stFeedoutPort.TableIndex].isFeedoutSideEnabled(stFeedoutPort.Side) THEN
								addToTargetFeedoutPorts(stFeedoutPort);
							END_IF
						END_FOR
					END_IF
					EXIT;
				END_IF
			END_FOR
		END_IF
		findAllEnabledFeedoutPorts := stDoorTrack.TargetFeedoutPorts.FeedoutPortsCount > 0;
	END_IF
END_IF
END_METHOD

METHOD findCandidateRoute : POINTER TO ST_Route
VAR_INPUT
	source : INT;
	target : INT;
END_VAR
VAR
	i : INT;
END_VAR
findCandidateRoute := 0;
FOR i:=0 TO MAIN.mainStateMachine.smCtrlInterface.config_stTransferTableConfig.PrimaryTable.RoutingTable.RoutesCount - 1 DO
	IF MAIN.mainStateMachine.smCtrlInterface.config_stTransferTableConfig.PrimaryTable.RoutingTable.Routes[i].SourceTableIndex = source AND
		MAIN.mainStateMachine.smCtrlInterface.config_stTransferTableConfig.PrimaryTable.RoutingTable.Routes[i].TargetTableIndex = target AND
		MAIN.mainStateMachine.smCtrlInterface.config_stTransferTableConfig.PrimaryTable.RoutingTable.Routes[i].PathsInfoCount > 0 THEN
		findCandidateRoute := ADR(MAIN.mainStateMachine.smCtrlInterface.config_stTransferTableConfig.PrimaryTable.RoutingTable.Routes[i]);
		RETURN;
	END_IF
END_FOR
END_METHOD

